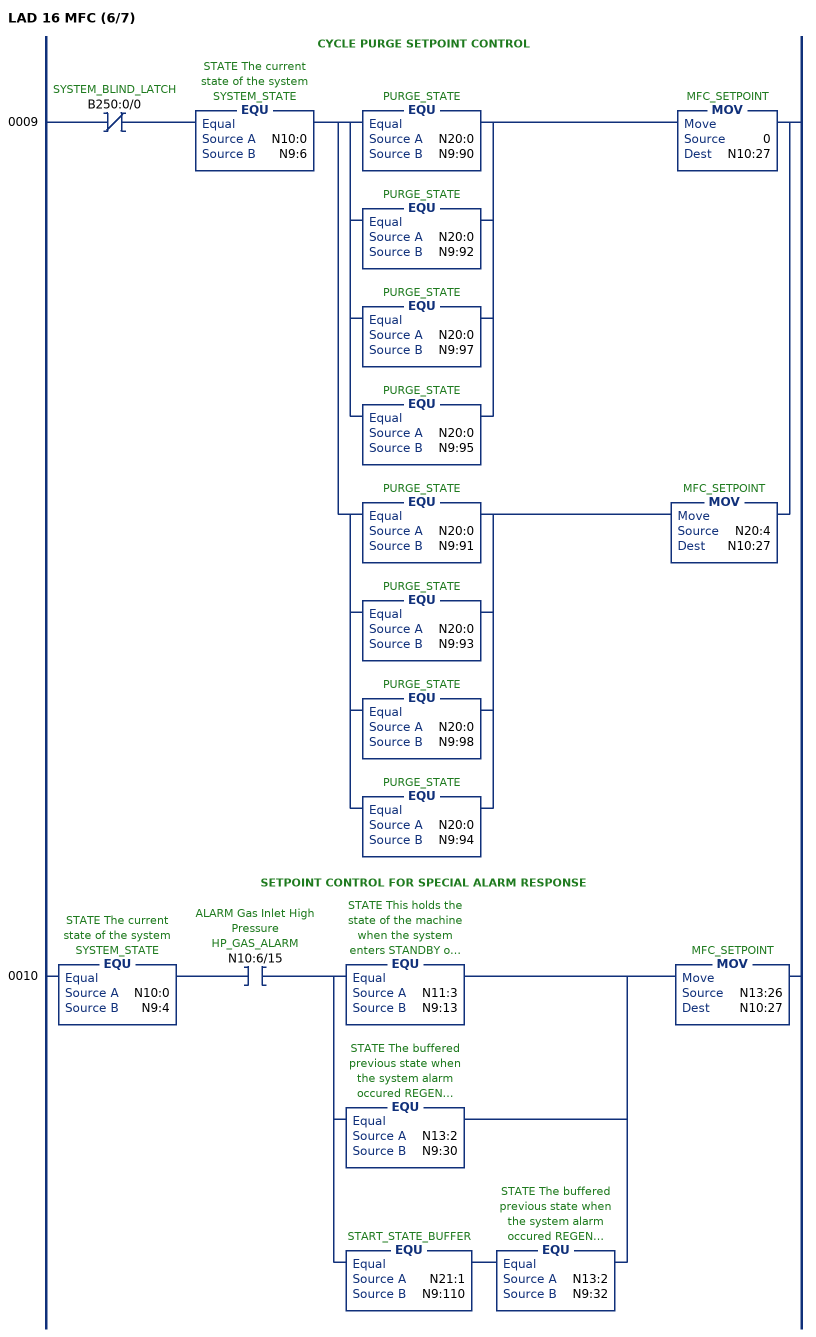
% Rung: 9 %
% TITLE: CYCLE PURGE SETPOINT CONTROL %
SOR XIO B250:0/0 EQU N10:0 N9:6 BST BST EQU N20:0 N9:90 NXB EQU N20:0 N9:92 NXB EQU N20:0 N9:97 NXB EQU N20:0 N9:95 BND MOV 0 N10:27 NXB BST EQU N20:0 N9:91 NXB EQU N20:0 N9:93 NXB EQU N20:0 N9:98 NXB EQU N20:0 N9:94 BND MOV N20:4 N10:27 BND EOR
%   B250:0/0  SYSTEM_BLIND_LATCH %
%   N10:0  SYSTEM_STATE  "STATE The current state of the system" %
%   N9:6  SYSTEM_PURGE %
%   N20:0  PURGE_STATE %
%   N9:90  PURGE_IDLE %
%   N9:92  PURGE_VENT_ADSORBER %
%   N9:97  PURGE_VENT_ADS_2 %
%   N9:95  PURGE_FINAL_VENT %
%   N10:27  MFC_SETPOINT %
%   N9:91  PURGE_INIT_VENT %
%   N9:93  PURGE_VENT_GETTER %
%   N9:98  PURGE_VENT_GET_2 %
%   N9:94  PURGE_BACKFILL %
%   N20:4  PURGE_FLOW %
% Rung: 10 %
% TITLE: SETPOINT CONTROL FOR SPECIAL ALARM RESPONSE %
SOR EQU N10:0 N9:4 XIC N10:6/15 BST EQU N11:3 N9:13 NXB EQU N13:2 N9:30 NXB EQU N21:1 N9:110 EQU N13:2 N9:32 BND MOV N13:26 N10:27 EOR
%   N10:0  SYSTEM_STATE  "STATE The current state of the system" %
%   N9:4  SYSTEM_ALARM  "STATE System Alarm" %
%   N10:6/15  HP_GAS_ALARM  "ALARM Gas Inlet High Pressure" %
%   N11:3  PROC_STATE_BUFFER  "STATE This holds the state of the machine when the system enters STANDBY or ALARM" %
%   N9:13  PROC_OVERLAP  "STATE Process Purify Overlap" %
%   N13:2  REGEN_SYSTEM_BUFFER  "STATE The buffered previous state when the system alarm occured" %
%   N9:30  REGEN_STANDBY  "STATE Regen Standby" %
%   N21:1  START_STATE_BUFFER %
%   N9:110  START_REG_VENT %
%   N9:32  REGEN_VENT  "STATE Regen Vent" %
%   N13:26  REGEN_BLEED_FLOW %
%   N10:27  MFC_SETPOINT %

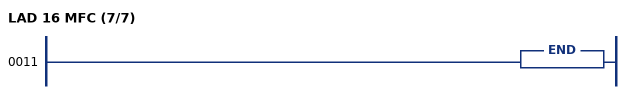
% Rung: 11 %
SOR END EOR

LADDER 17 "BYPASS"    % Controls the bypass %
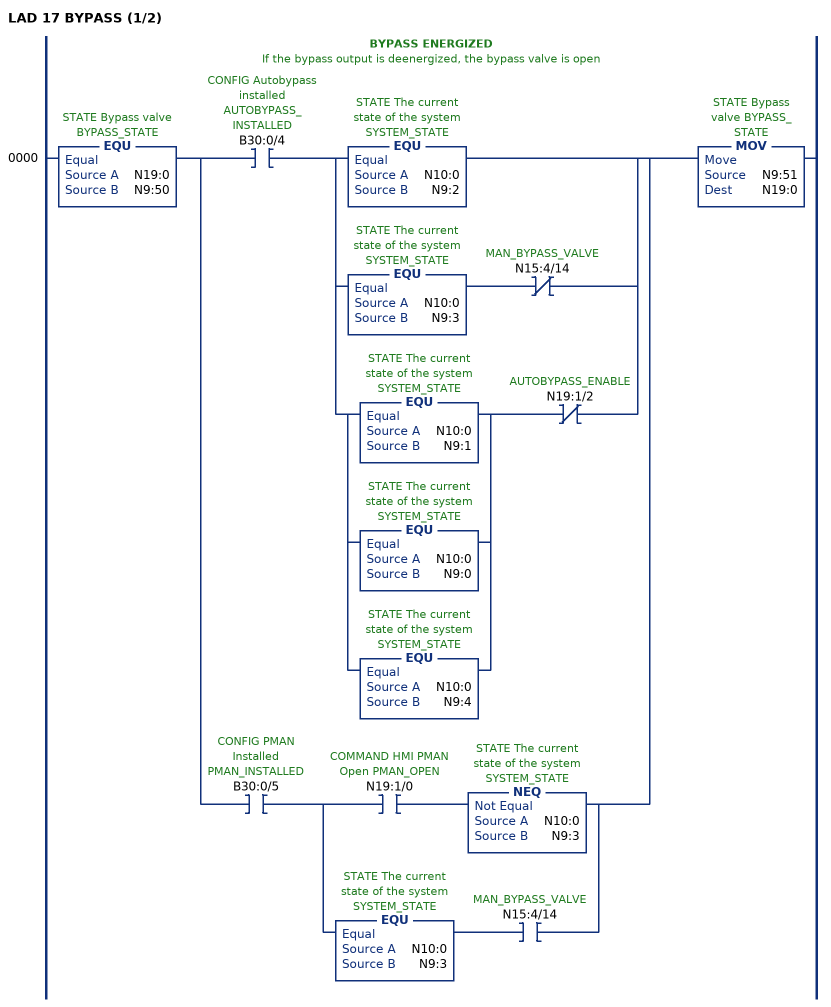
% Rung: 0 %
% TITLE: BYPASS ENERGIZED %
% If the bypass output is deenergized, the bypass valve is open %
SOR EQU N19:0 N9:50 BST XIC B30:0/4 BST EQU N10:0 N9:2 NXB EQU N10:0 N9:3 XIO N15:4/14 NXB BST EQU N10:0 N9:1 NXB EQU N10:0 N9:0 NXB EQU N10:0 N9:4 BND XIO N19:1/2 BND NXB XIC B30:0/5 BST XIC N19:1/0 NEQ N10:0 N9:3 NXB EQU N10:0 N9:3 XIC N15:4/14 BND BND MOV N9:51 N19:0 EOR
%   N19:0  BYPASS_STATE  "STATE Bypass valve" %
%   N9:50  BYPASS_DEENERGIZED  "STATE Bypass Deenergized" %
%   B30:0/4  AUTOBYPASS_INSTALLED  "CONFIG Autobypass installed" %
%   N10:0  SYSTEM_STATE  "STATE The current state of the system" %
%   N9:2  SYSTEM_PROCESS  "STATE System Process" %
%   N9:3  SYSTEM_MANUAL  "STATE System Manual" %
%   N15:4/14  MAN_BYPASS_VALVE %
%   N9:1  SYSTEM_STANDBY  "STATE System Process" %
%   N9:0  SYSTEM_OFFLINE %
%   N9:4  SYSTEM_ALARM  "STATE System Alarm" %
%   N19:1/2  AUTOBYPASS_ENABLE %
%   B30:0/5  PMAN_INSTALLED  "CONFIG PMAN Installed" %
%   N19:1/0  PMAN_OPEN  "COMMAND HMI PMAN Open" %
%   N9:51  BYPASS_ENERGIZED  "STATE Bypass Energized" %

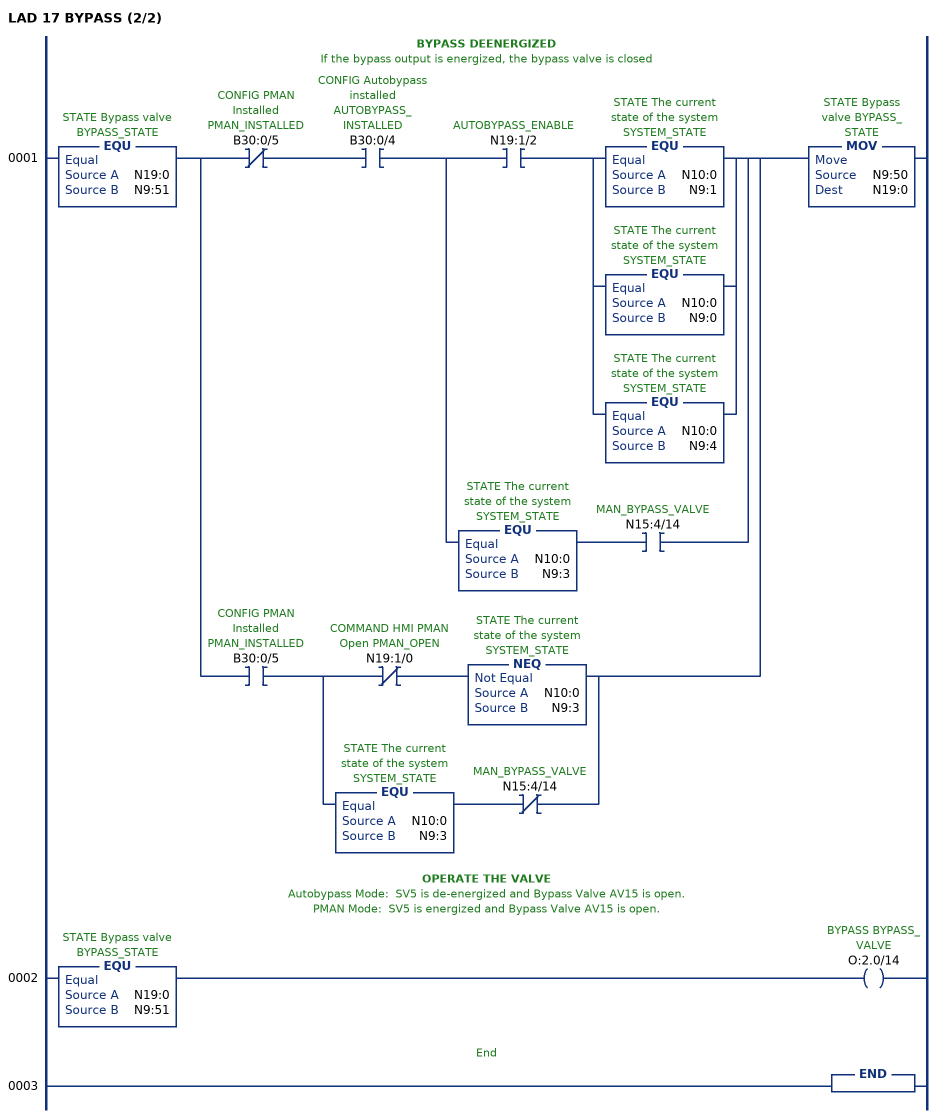
% Rung: 1 %
% TITLE: BYPASS DEENERGIZED %
% If the bypass output is energized, the bypass valve is closed %
SOR EQU N19:0 N9:51 BST XIO B30:0/5 XIC B30:0/4 BST XIC N19:1/2 BST EQU N10:0 N9:1 NXB EQU N10:0 N9:0 NXB EQU N10:0 N9:4 BND NXB EQU N10:0 N9:3 XIC N15:4/14 BND NXB XIC B30:0/5 BST XIO N19:1/0 NEQ N10:0 N9:3 NXB EQU N10:0 N9:3 XIO N15:4/14 BND BND MOV N9:50 N19:0 EOR
%   N19:0  BYPASS_STATE  "STATE Bypass valve" %
%   N9:51  BYPASS_ENERGIZED  "STATE Bypass Energized" %
%   B30:0/5  PMAN_INSTALLED  "CONFIG PMAN Installed" %
%   B30:0/4  AUTOBYPASS_INSTALLED  "CONFIG Autobypass installed" %
%   N19:1/2  AUTOBYPASS_ENABLE %
%   N10:0  SYSTEM_STATE  "STATE The current state of the system" %
%   N9:1  SYSTEM_STANDBY  "STATE System Process" %
%   N9:0  SYSTEM_OFFLINE %
%   N9:4  SYSTEM_ALARM  "STATE System Alarm" %
%   N9:3  SYSTEM_MANUAL  "STATE System Manual" %
%   N15:4/14  MAN_BYPASS_VALVE %
%   N19:1/0  PMAN_OPEN  "COMMAND HMI PMAN Open" %
%   N9:50  BYPASS_DEENERGIZED  "STATE Bypass Deenergized" %
% Rung: 2 %
% TITLE: OPERATE THE VALVE %
% Autobypass Mode:  SV5 is de-energized and Bypass Valve AV15 is open.
% PMAN Mode:  SV5 is energized and Bypass Valve AV15 is open. %
SOR EQU N19:0 N9:51 OTE O:2.0/14 EOR
%   N19:0  BYPASS_STATE  "STATE Bypass valve" %
%   N9:51  BYPASS_ENERGIZED  "STATE Bypass Energized" %
%   O:2.0/14  BYPASS_VALVE  "BYPASS" %
% Rung: 3 %
% End %
SOR END EOR

LADDER 20 "ADS A"    % Controls the Adsorber A %
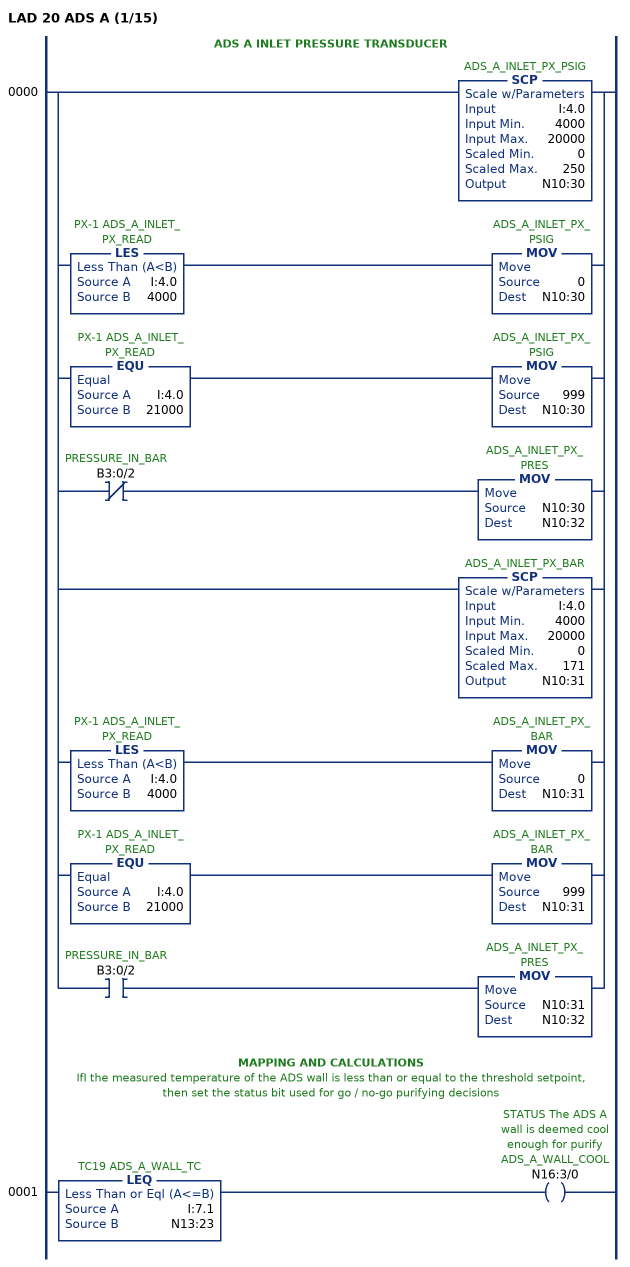
% Rung: 0 %
% TITLE: ADS A INLET PRESSURE TRANSDUCER %
SOR BST SCP I:4.0 4000 20000 0 250 N10:30 NXB LES I:4.0 4000 MOV 0 N10:30 NXB EQU I:4.0 21000 MOV 999 N10:30 NXB XIO B3:0/2 MOV N10:30 N10:32 NXB SCP I:4.0 4000 20000 0 171 N10:31 NXB LES I:4.0 4000 MOV 0 N10:31 NXB EQU I:4.0 21000 MOV 999 N10:31 NXB XIC B3:0/2 MOV N10:31 N10:32 BND EOR
%   I:4.0  ADS_A_INLET_PX_READ  "PX-1" %
%   N10:30  ADS_A_INLET_PX_PSIG %
%   B3:0/2  PRESSURE_IN_BAR %
%   N10:32  ADS_A_INLET_PX_PRES %
%   N10:31  ADS_A_INLET_PX_BAR %
% Rung: 1 %
% TITLE: MAPPING AND CALCULATIONS %
% IfI the measured temperature of the ADS wall is less than or equal to the threshold setpoint, then set the status bit used for go / no-go purifying decisions %
SOR LEQ I:7.1 N13:23 OTE N16:3/0 EOR
%   I:7.1  ADS_A_WALL_TC  "TC19" %
%   N13:23  ADS_WALL_TEMP_COOL  "CONFIG The temp at which the adsorber wall is deemed to be cool enough to purify" %
%   N16:3/0  ADS_A_WALL_COOL  "STATUS The ADS A wall is deemed cool enough for purify" %

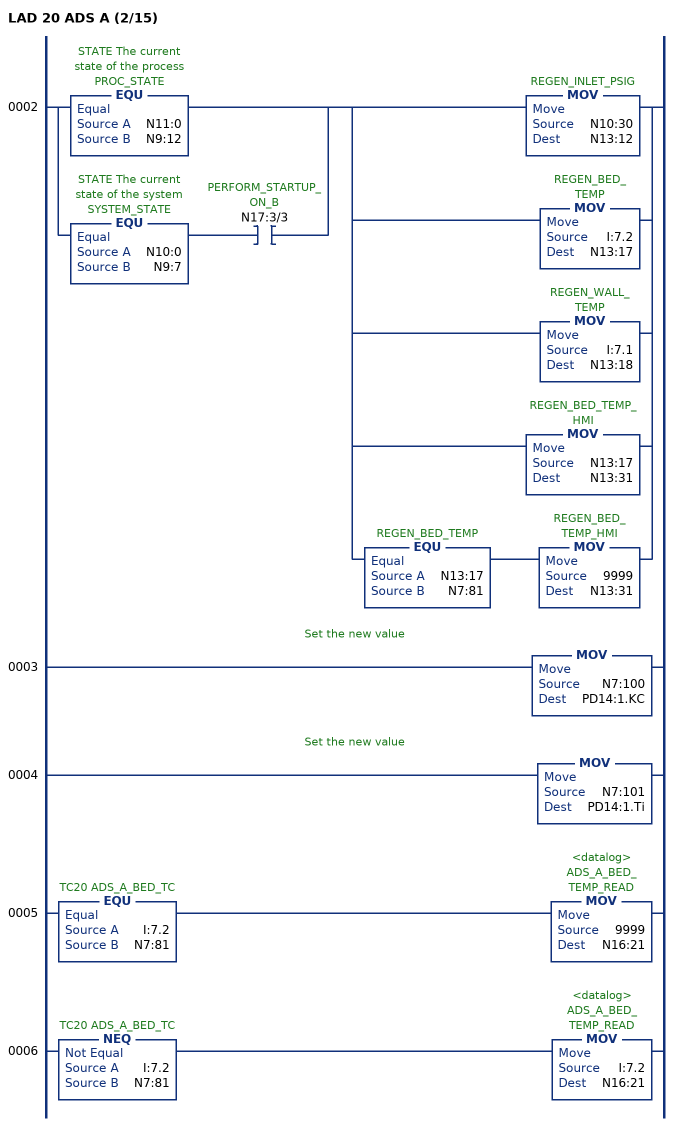
% Rung: 2 %
SOR BST EQU N11:0 N9:12 NXB EQU N10:0 N9:7 XIC N17:3/3 BND BST MOV N10:30 N13:12 NXB MOV I:7.2 N13:17 NXB MOV I:7.1 N13:18 NXB MOV N13:17 N13:31 NXB EQU N13:17 N7:81 MOV 9999 N13:31 BND EOR
%   N11:0  PROC_STATE  "STATE The current state of the process" %
%   N9:12  PROC_PFY_B_REG_A  "STATE Process Purify B" %
%   N10:0  SYSTEM_STATE  "STATE The current state of the system" %
%   N9:7  SYSTEM_COLD_START %
%   N17:3/3  PERFORM_STARTUP_ON_B %
%   N10:30  ADS_A_INLET_PX_PSIG %
%   N13:12  REGEN_INLET_PSIG %
%   I:7.2  ADS_A_BED_TC  "TC20" %
%   N13:17  REGEN_BED_TEMP %
%   I:7.1  ADS_A_WALL_TC  "TC19" %
%   N13:18  REGEN_WALL_TEMP %
%   N13:31  REGEN_BED_TEMP_HMI %
%   N7:81  TC_OPEN_SP  "CONFIG The value read by an open TC input" %
% Rung: 3 %
% Set the new value %
SOR MOV N7:100 PD14:1.KC EOR
%   N7:100  BLANKET_P  "CONFIG Blanket Proportional Gain New" %
% Rung: 4 %
% Set the new value %
SOR MOV N7:101 PD14:1.Ti EOR
%   N7:101  BLANKET_I  "CONFIG Blanket Integral Gain New" %
% Rung: 5 %
SOR EQU I:7.2 N7:81 MOV 9999 N16:21 EOR
%   I:7.2  ADS_A_BED_TC  "TC20" %
%   N7:81  TC_OPEN_SP  "CONFIG The value read by an open TC input" %
%   N16:21  ADS_A_BED_TEMP_READ  "<datalog>" %
% Rung: 6 %
SOR NEQ I:7.2 N7:81 MOV I:7.2 N16:21 EOR
%   I:7.2  ADS_A_BED_TC  "TC20" %
%   N7:81  TC_OPEN_SP  "CONFIG The value read by an open TC input" %
%   N16:21  ADS_A_BED_TEMP_READ  "<datalog>" %

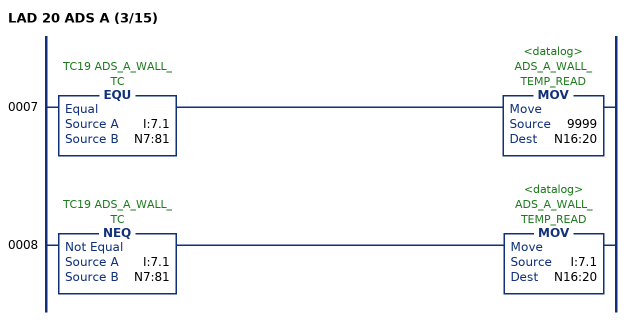
% Rung: 7 %
SOR EQU I:7.1 N7:81 MOV 9999 N16:20 EOR
%   I:7.1  ADS_A_WALL_TC  "TC19" %
%   N7:81  TC_OPEN_SP  "CONFIG The value read by an open TC input" %
%   N16:20  ADS_A_WALL_TEMP_READ  "<datalog>" %
% Rung: 8 %
SOR NEQ I:7.1 N7:81 MOV I:7.1 N16:20 EOR
%   I:7.1  ADS_A_WALL_TC  "TC19" %
%   N7:81  TC_OPEN_SP  "CONFIG The value read by an open TC input" %
%   N16:20  ADS_A_WALL_TEMP_READ  "<datalog>" %

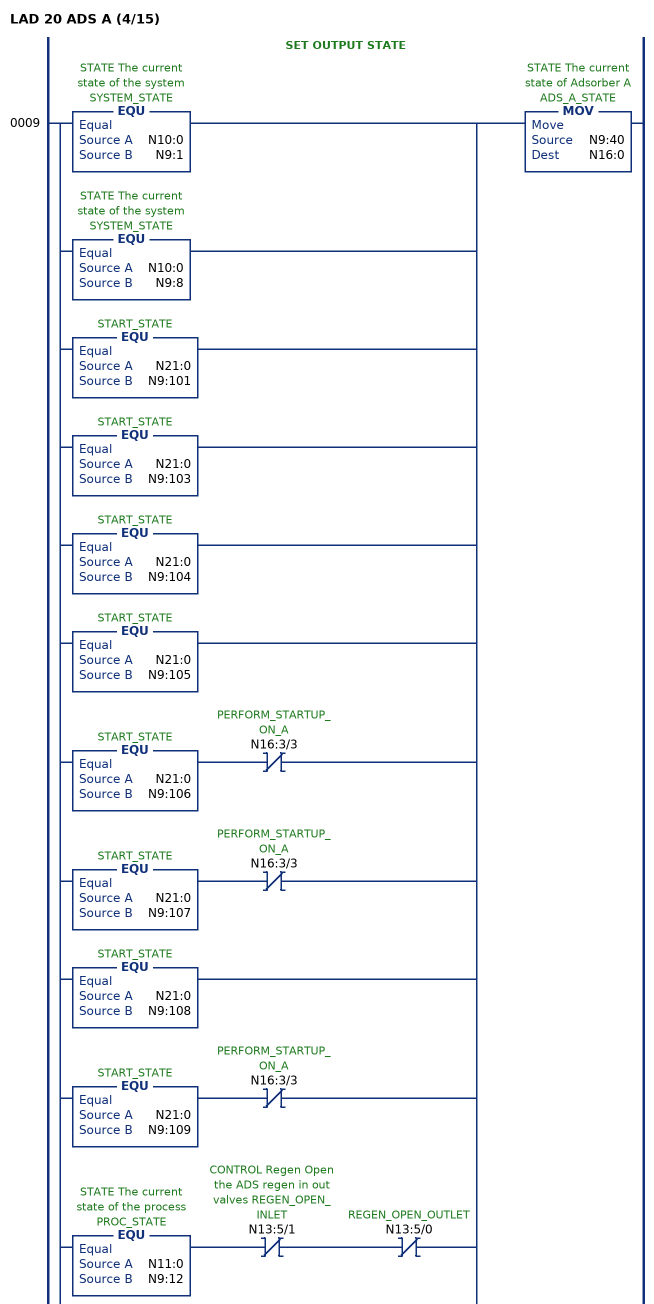

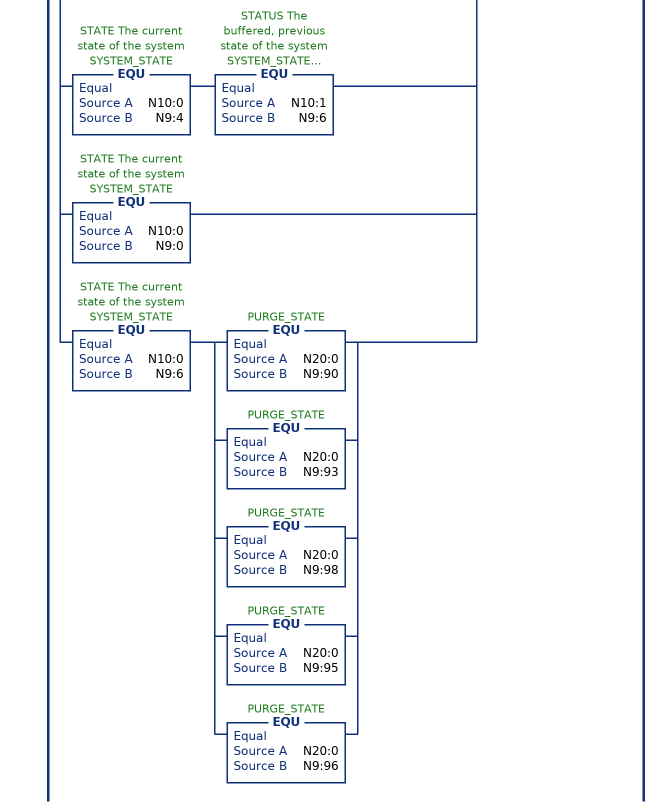
% Rung: 9 %
% TITLE: SET OUTPUT STATE %
SOR BST EQU N10:0 N9:1 NXB EQU N10:0 N9:8 NXB BST EQU N21:0 N9:101 NXB EQU N21:0 N9:103 NXB EQU N21:0 N9:104 NXB EQU N21:0 N9:105 NXB EQU N21:0 N9:106 XIO N16:3/3 NXB EQU N21:0 N9:107 XIO N16:3/3 NXB EQU N21:0 N9:108 NXB EQU N21:0 N9:109 XIO N16:3/3 BND NXB EQU N11:0 N9:12 XIO N13:5/1 XIO N13:5/0 NXB EQU N10:0 N9:4 EQU N10:1 N9:6 NXB EQU N10:0 N9:0 NXB EQU N10:0 N9:6 BST EQU N20:0 N9:90 NXB EQU N20:0 N9:93 NXB EQU N20:0 N9:98 NXB EQU N20:0 N9:95 NXB EQU N20:0 N9:96 BND BND MOV N9:40 N16:0 EOR
%   N10:0  SYSTEM_STATE  "STATE The current state of the system" %
%   N9:1  SYSTEM_STANDBY  "STATE System Process" %
%   N9:8  SYSTEM_SUPPLEMENTAL %
%   N21:0  START_STATE %
%   N9:101  START_COOL %
%   N9:103  START_VENT_GET_1 %
%   N9:104  START_HEAT %
%   N9:105  START_VENT_ALL %
%   N9:106  START_BACKFILL_1 %
%   N16:3/3  PERFORM_STARTUP_ON_A %
%   N9:107  START_VENT_ADS_2 %
%   N9:108  START_VENT_GET_2 %
%   N9:109  START_BACKFILL_2 %
%   N11:0  PROC_STATE  "STATE The current state of the process" %
%   N9:12  PROC_PFY_B_REG_A  "STATE Process Purify B" %
%   N13:5/1  REGEN_OPEN_INLET  "CONTROL Regen Open the ADS regen in out valves" %
%   N13:5/0  REGEN_OPEN_OUTLET %
%   N9:4  SYSTEM_ALARM  "STATE System Alarm" %
%   N10:1  SYSTEM_STATE_BUFFER  "STATUS The buffered, previous state of the system" %
%   N9:6  SYSTEM_PURGE %
%   N9:0  SYSTEM_OFFLINE %
%   N20:0  PURGE_STATE %
%   N9:90  PURGE_IDLE %
%   N9:93  PURGE_VENT_GETTER %
%   N9:98  PURGE_VENT_GET_2 %
%   N9:95  PURGE_FINAL_VENT %
%   N9:96  PURGE_DONE %
%   N9:40  ADS_STANDBY  "STATE ADS Standby" %
%   N16:0  ADS_A_STATE  "STATE The current state of Adsorber A" %

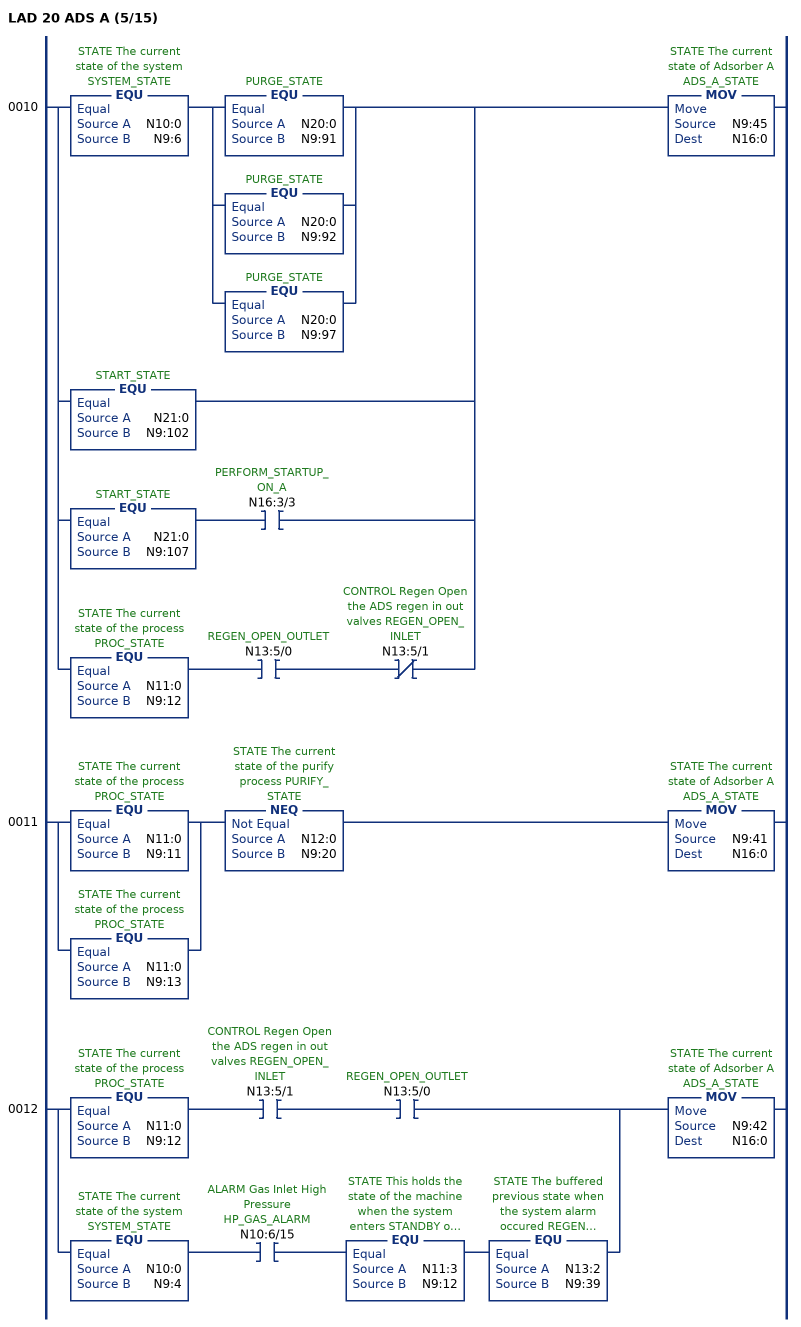
% Rung: 10 %
SOR BST EQU N10:0 N9:6 BST EQU N20:0 N9:91 NXB EQU N20:0 N9:92 NXB EQU N20:0 N9:97 BND NXB BST EQU N21:0 N9:102 NXB EQU N21:0 N9:107 XIC N16:3/3 BND NXB EQU N11:0 N9:12 XIC N13:5/0 XIO N13:5/1 BND MOV N9:45 N16:0 EOR
%   N10:0  SYSTEM_STATE  "STATE The current state of the system" %
%   N9:6  SYSTEM_PURGE %
%   N20:0  PURGE_STATE %
%   N9:91  PURGE_INIT_VENT %
%   N9:92  PURGE_VENT_ADSORBER %
%   N9:97  PURGE_VENT_ADS_2 %
%   N21:0  START_STATE %
%   N9:102  START_VENT_ADS_1 %
%   N9:107  START_VENT_ADS_2 %
%   N16:3/3  PERFORM_STARTUP_ON_A %
%   N11:0  PROC_STATE  "STATE The current state of the process" %
%   N9:12  PROC_PFY_B_REG_A  "STATE Process Purify B" %
%   N13:5/0  REGEN_OPEN_OUTLET %
%   N13:5/1  REGEN_OPEN_INLET  "CONTROL Regen Open the ADS regen in out valves" %
%   N9:45  ADS_VENT %
%   N16:0  ADS_A_STATE  "STATE The current state of Adsorber A" %
% Rung: 11 %
SOR BST EQU N11:0 N9:11 NXB EQU N11:0 N9:13 BND NEQ N12:0 N9:20 MOV N9:41 N16:0 EOR
%   N11:0  PROC_STATE  "STATE The current state of the process" %
%   N9:11  PROC_PFY_A_REG_B  "STATE Process Purify A" %
%   N9:13  PROC_OVERLAP  "STATE Process Purify Overlap" %
%   N12:0  PURIFY_STATE  "STATE The current state of the purify process" %
%   N9:20  PURIFY_STANDBY  "STATE Purify Standby" %
%   N9:41  ADS_PURIFY  "STATE ADS Purify" %
%   N16:0  ADS_A_STATE  "STATE The current state of Adsorber A" %
% Rung: 12 %
SOR BST EQU N11:0 N9:12 XIC N13:5/1 XIC N13:5/0 NXB EQU N10:0 N9:4 XIC N10:6/15 EQU N11:3 N9:12 EQU N13:2 N9:39 BND MOV N9:42 N16:0 EOR
%   N11:0  PROC_STATE  "STATE The current state of the process" %
%   N9:12  PROC_PFY_B_REG_A  "STATE Process Purify B" %
%   N13:5/1  REGEN_OPEN_INLET  "CONTROL Regen Open the ADS regen in out valves" %
%   N13:5/0  REGEN_OPEN_OUTLET %
%   N10:0  SYSTEM_STATE  "STATE The current state of the system" %
%   N9:4  SYSTEM_ALARM  "STATE System Alarm" %
%   N10:6/15  HP_GAS_ALARM  "ALARM Gas Inlet High Pressure" %
%   N11:3  PROC_STATE_BUFFER  "STATE This holds the state of the machine when the system enters STANDBY or ALARM" %
%   N13:2  REGEN_SYSTEM_BUFFER  "STATE The buffered previous state when the system alarm occured" %
%   N9:39  REGEN_BACKFILL %
%   N9:42  ADS_REGEN  "STATE ADS Regen" %
%   N16:0  ADS_A_STATE  "STATE The current state of Adsorber A" %

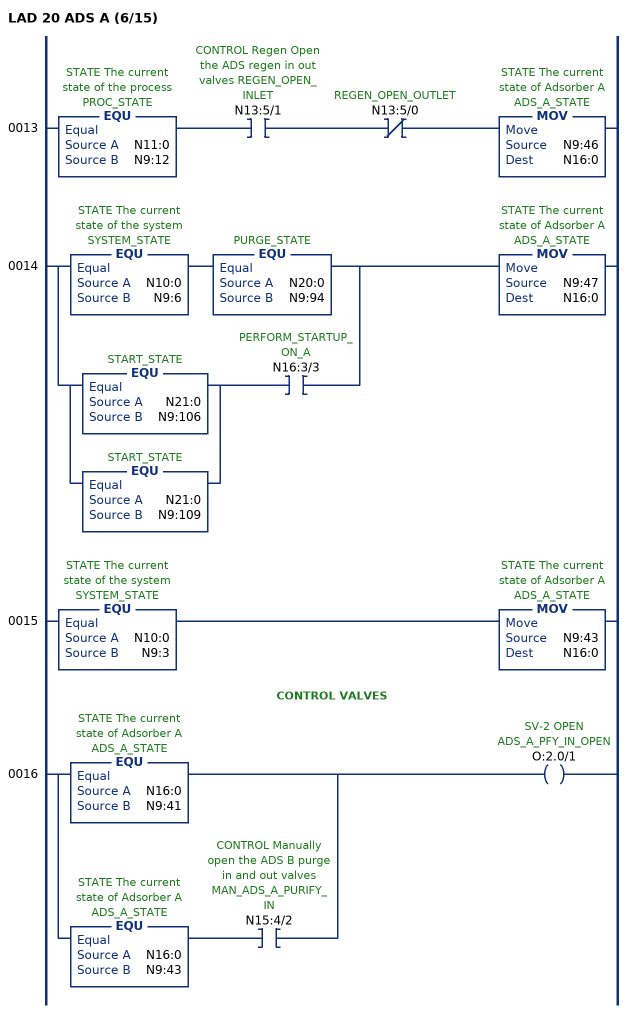
% Rung: 13 %
SOR EQU N11:0 N9:12 XIC N13:5/1 XIO N13:5/0 MOV N9:46 N16:0 EOR
%   N11:0  PROC_STATE  "STATE The current state of the process" %
%   N9:12  PROC_PFY_B_REG_A  "STATE Process Purify B" %
%   N13:5/1  REGEN_OPEN_INLET  "CONTROL Regen Open the ADS regen in out valves" %
%   N13:5/0  REGEN_OPEN_OUTLET %
%   N9:46  ADS_REGEN_BACKFILL %
%   N16:0  ADS_A_STATE  "STATE The current state of Adsorber A" %
% Rung: 14 %
SOR BST EQU N10:0 N9:6 EQU N20:0 N9:94 NXB BST EQU N21:0 N9:106 NXB EQU N21:0 N9:109 BND XIC N16:3/3 BND MOV N9:47 N16:0 EOR
%   N10:0  SYSTEM_STATE  "STATE The current state of the system" %
%   N9:6  SYSTEM_PURGE %
%   N20:0  PURGE_STATE %
%   N9:94  PURGE_BACKFILL %
%   N21:0  START_STATE %
%   N9:106  START_BACKFILL_1 %
%   N9:109  START_BACKFILL_2 %
%   N16:3/3  PERFORM_STARTUP_ON_A %
%   N9:47  ADS_BACKFILL %
%   N16:0  ADS_A_STATE  "STATE The current state of Adsorber A" %
% Rung: 15 %
SOR EQU N10:0 N9:3 MOV N9:43 N16:0 EOR
%   N10:0  SYSTEM_STATE  "STATE The current state of the system" %
%   N9:3  SYSTEM_MANUAL  "STATE System Manual" %
%   N9:43  ADS_MANUAL  "STATE ADS Manual" %
%   N16:0  ADS_A_STATE  "STATE The current state of Adsorber A" %
% Rung: 16 %
% TITLE: CONTROL VALVES %
SOR BST EQU N16:0 N9:41 NXB EQU N16:0 N9:43 XIC N15:4/2 BND OTE O:2.0/1 EOR
%   N16:0  ADS_A_STATE  "STATE The current state of Adsorber A" %
%   N9:41  ADS_PURIFY  "STATE ADS Purify" %
%   N9:43  ADS_MANUAL  "STATE ADS Manual" %
%   N15:4/2  MAN_ADS_A_PURIFY_IN  "CONTROL Manually open the ADS B purge in and out valves" %
%   O:2.0/1  ADS_A_PFY_IN_OPEN  "SV-2 OPEN" %

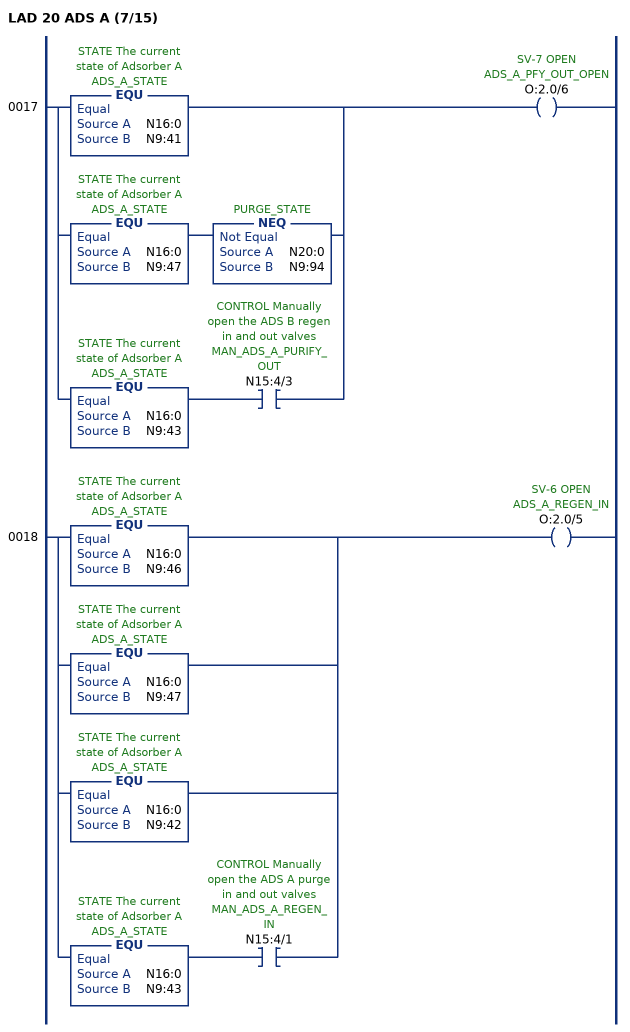
% Rung: 17 %
SOR BST EQU N16:0 N9:41 NXB EQU N16:0 N9:47 NEQ N20:0 N9:94 NXB EQU N16:0 N9:43 XIC N15:4/3 BND OTE O:2.0/6 EOR
%   N16:0  ADS_A_STATE  "STATE The current state of Adsorber A" %
%   N9:41  ADS_PURIFY  "STATE ADS Purify" %
%   N9:47  ADS_BACKFILL %
%   N20:0  PURGE_STATE %
%   N9:94  PURGE_BACKFILL %
%   N9:43  ADS_MANUAL  "STATE ADS Manual" %
%   N15:4/3  MAN_ADS_A_PURIFY_OUT  "CONTROL Manually open the ADS B regen in and out valves" %
%   O:2.0/6  ADS_A_PFY_OUT_OPEN  "SV-7 OPEN" %
% Rung: 18 %
SOR BST EQU N16:0 N9:46 NXB EQU N16:0 N9:47 NXB EQU N16:0 N9:42 NXB EQU N16:0 N9:43 XIC N15:4/1 BND OTE O:2.0/5 EOR
%   N16:0  ADS_A_STATE  "STATE The current state of Adsorber A" %
%   N9:46  ADS_REGEN_BACKFILL %
%   N9:47  ADS_BACKFILL %
%   N9:42  ADS_REGEN  "STATE ADS Regen" %
%   N9:43  ADS_MANUAL  "STATE ADS Manual" %
%   N15:4/1  MAN_ADS_A_REGEN_IN  "CONTROL Manually open the ADS A purge in and out valves" %
%   O:2.0/5  ADS_A_REGEN_IN  "SV-6 OPEN" %

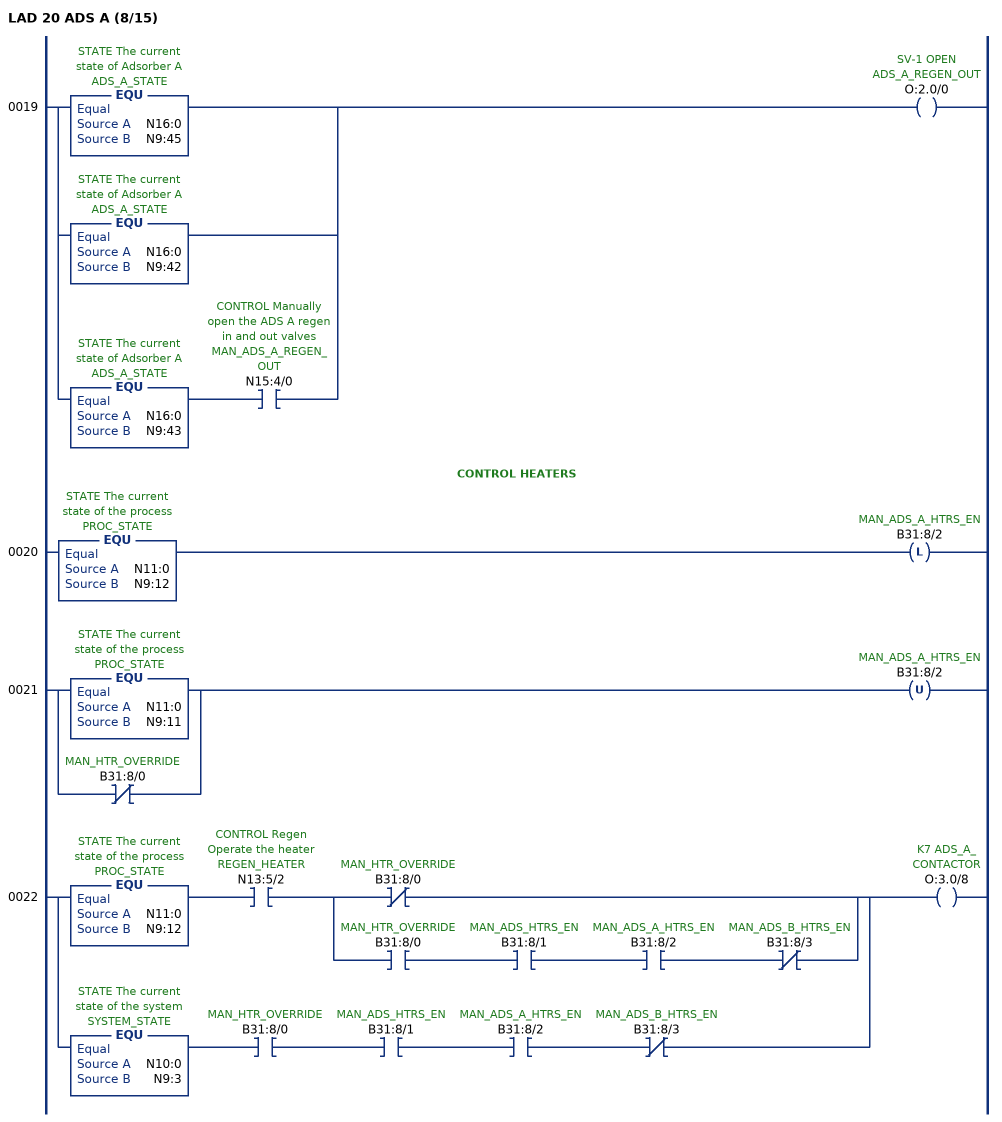
% Rung: 19 %
SOR BST EQU N16:0 N9:45 NXB EQU N16:0 N9:42 NXB EQU N16:0 N9:43 XIC N15:4/0 BND OTE O:2.0/0 EOR
%   N16:0  ADS_A_STATE  "STATE The current state of Adsorber A" %
%   N9:45  ADS_VENT %
%   N9:42  ADS_REGEN  "STATE ADS Regen" %
%   N9:43  ADS_MANUAL  "STATE ADS Manual" %
%   N15:4/0  MAN_ADS_A_REGEN_OUT  "CONTROL Manually open the ADS A regen in and out valves" %
%   O:2.0/0  ADS_A_REGEN_OUT  "SV-1 OPEN" %
% Rung: 20 %
% TITLE: CONTROL HEATERS %
SOR EQU N11:0 N9:12 OTL B31:8/2 EOR
%   N11:0  PROC_STATE  "STATE The current state of the process" %
%   N9:12  PROC_PFY_B_REG_A  "STATE Process Purify B" %
%   B31:8/2  MAN_ADS_A_HTRS_EN %
% Rung: 21 %
SOR BST EQU N11:0 N9:11 NXB XIO B31:8/0 BND OTU B31:8/2 EOR
%   N11:0  PROC_STATE  "STATE The current state of the process" %
%   N9:11  PROC_PFY_A_REG_B  "STATE Process Purify A" %
%   B31:8/0  MAN_HTR_OVERRIDE %
%   B31:8/2  MAN_ADS_A_HTRS_EN %
% Rung: 22 %
SOR BST EQU N11:0 N9:12 XIC N13:5/2 BST XIO B31:8/0 NXB XIC B31:8/0 XIC B31:8/1 XIC B31:8/2 XIO B31:8/3 BND NXB EQU N10:0 N9:3 XIC B31:8/0 XIC B31:8/1 XIC B31:8/2 XIO B31:8/3 BND OTE O:3.0/8 EOR
%   N11:0  PROC_STATE  "STATE The current state of the process" %
%   N9:12  PROC_PFY_B_REG_A  "STATE Process Purify B" %
%   N13:5/2  REGEN_HEATER  "CONTROL Regen Operate the heater" %
%   B31:8/0  MAN_HTR_OVERRIDE %
%   B31:8/1  MAN_ADS_HTRS_EN %
%   B31:8/2  MAN_ADS_A_HTRS_EN %
%   B31:8/3  MAN_ADS_B_HTRS_EN %
%   N10:0  SYSTEM_STATE  "STATE The current state of the system" %
%   N9:3  SYSTEM_MANUAL  "STATE System Manual" %
%   O:3.0/8  ADS_A_CONTACTOR  "K7" %

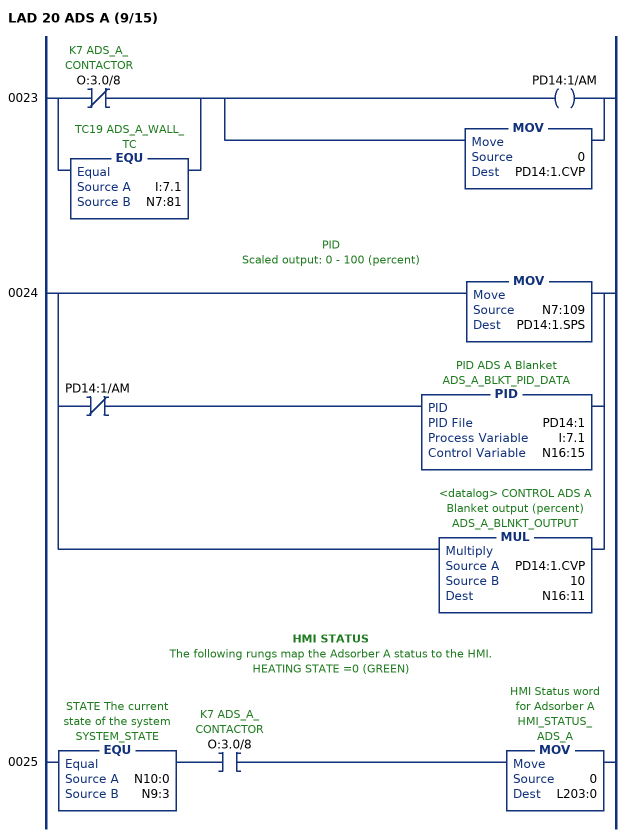
% Rung: 23 %
SOR BST XIO O:3.0/8 NXB EQU I:7.1 N7:81 BND BST OTE PD14:1/AM NXB MOV 0 PD14:1.CVP BND EOR
%   O:3.0/8  ADS_A_CONTACTOR  "K7" %
%   I:7.1  ADS_A_WALL_TC  "TC19" %
%   N7:81  TC_OPEN_SP  "CONFIG The value read by an open TC input" %
% Rung: 24 %
% PID
% Scaled output: 0 - 100 (percent) %
SOR BST MOV N7:109 PD14:1.SPS NXB XIO PD14:1/AM PID PD14:1 I:7.1 N16:15 NXB MUL PD14:1.CVP 10 N16:11 BND EOR
%   N7:109  BLANKET_SP  "<datalog> CONTROL Blanket PID Setpoint" %
%   PD14:1  ADS_A_BLKT_PID_DATA  "PID ADS A Blanket" %
%   I:7.1  ADS_A_WALL_TC  "TC19" %
%   N16:15  ADS_A_BLKT_OUTPT_RAW  "CONTROL ADS A Blanket PID Output Raw" %
%   N16:11  ADS_A_BLNKT_OUTPUT  "<datalog> CONTROL ADS A Blanket output (percent)" %
% Rung: 25 %
% TITLE: HMI STATUS %
% The following rungs map the Adsorber A status to the HMI.
% HEATING STATE =0 (GREEN) %
SOR EQU N10:0 N9:3 XIC O:3.0/8 MOV 0 L203:0 EOR
%   N10:0  SYSTEM_STATE  "STATE The current state of the system" %
%   N9:3  SYSTEM_MANUAL  "STATE System Manual" %
%   O:3.0/8  ADS_A_CONTACTOR  "K7" %
%   L203:0  HMI_STATUS_ADS_A  "HMI Status word for Adsorber A" %

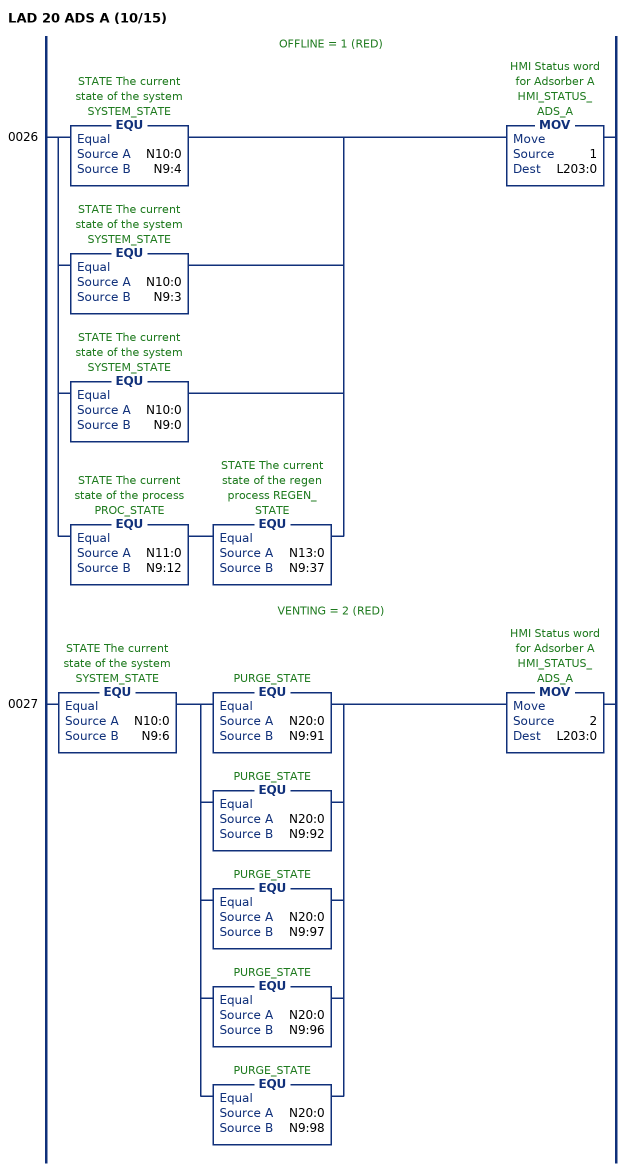
% Rung: 26 %
% OFFLINE = 1 (RED) %
SOR BST BST EQU N10:0 N9:4 NXB EQU N10:0 N9:3 NXB EQU N10:0 N9:0 BND NXB EQU N11:0 N9:12 EQU N13:0 N9:37 BND MOV 1 L203:0 EOR
%   N10:0  SYSTEM_STATE  "STATE The current state of the system" %
%   N9:4  SYSTEM_ALARM  "STATE System Alarm" %
%   N9:3  SYSTEM_MANUAL  "STATE System Manual" %
%   N9:0  SYSTEM_OFFLINE %
%   N11:0  PROC_STATE  "STATE The current state of the process" %
%   N9:12  PROC_PFY_B_REG_A  "STATE Process Purify B" %
%   N13:0  REGEN_STATE  "STATE The current state of the regen process" %
%   N9:37  REGEN_ALARM  "STATE Regen Alarm" %
%   L203:0  HMI_STATUS_ADS_A  "HMI Status word for Adsorber A" %
% Rung: 27 %
% VENTING = 2 (RED) %
SOR EQU N10:0 N9:6 BST EQU N20:0 N9:91 NXB EQU N20:0 N9:92 NXB EQU N20:0 N9:97 NXB EQU N20:0 N9:96 NXB EQU N20:0 N9:98 BND MOV 2 L203:0 EOR
%   N10:0  SYSTEM_STATE  "STATE The current state of the system" %
%   N9:6  SYSTEM_PURGE %
%   N20:0  PURGE_STATE %
%   N9:91  PURGE_INIT_VENT %
%   N9:92  PURGE_VENT_ADSORBER %
%   N9:97  PURGE_VENT_ADS_2 %
%   N9:96  PURGE_DONE %
%   N9:98  PURGE_VENT_GET_2 %
%   L203:0  HMI_STATUS_ADS_A  "HMI Status word for Adsorber A" %

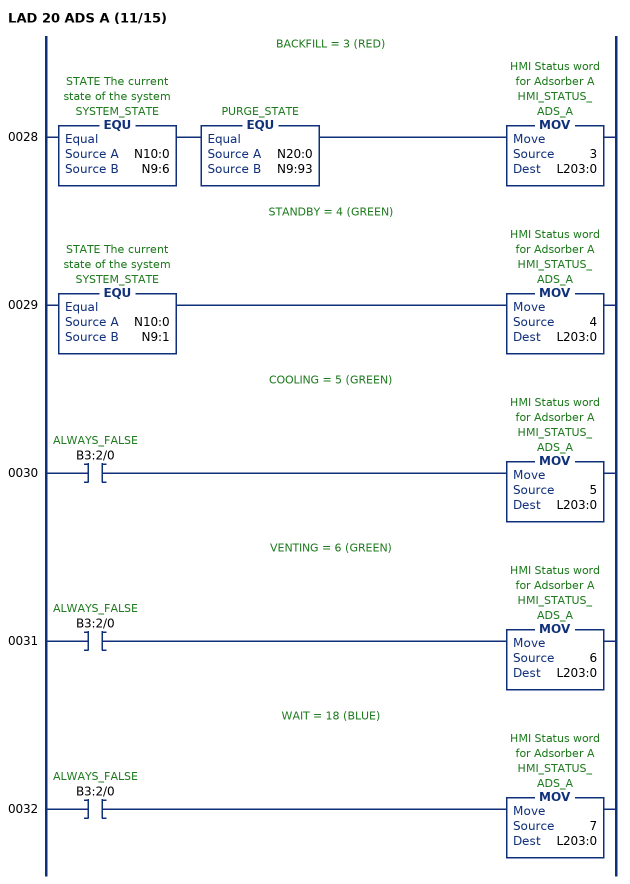
% Rung: 28 %
% BACKFILL = 3 (RED) %
SOR EQU N10:0 N9:6 EQU N20:0 N9:93 MOV 3 L203:0 EOR
%   N10:0  SYSTEM_STATE  "STATE The current state of the system" %
%   N9:6  SYSTEM_PURGE %
%   N20:0  PURGE_STATE %
%   N9:93  PURGE_VENT_GETTER %
%   L203:0  HMI_STATUS_ADS_A  "HMI Status word for Adsorber A" %
% Rung: 29 %
% STANDBY = 4 (GREEN) %
SOR EQU N10:0 N9:1 MOV 4 L203:0 EOR
%   N10:0  SYSTEM_STATE  "STATE The current state of the system" %
%   N9:1  SYSTEM_STANDBY  "STATE System Process" %
%   L203:0  HMI_STATUS_ADS_A  "HMI Status word for Adsorber A" %
% Rung: 30 %
% COOLING = 5 (GREEN) %
SOR XIC B3:2/0 MOV 5 L203:0 EOR
%   B3:2/0  ALWAYS_FALSE %
%   L203:0  HMI_STATUS_ADS_A  "HMI Status word for Adsorber A" %
% Rung: 31 %
% VENTING = 6 (GREEN) %
SOR XIC B3:2/0 MOV 6 L203:0 EOR
%   B3:2/0  ALWAYS_FALSE %
%   L203:0  HMI_STATUS_ADS_A  "HMI Status word for Adsorber A" %
% Rung: 32 %
% WAIT = 18 (BLUE) %
SOR XIC B3:2/0 MOV 7 L203:0 EOR
%   B3:2/0  ALWAYS_FALSE %
%   L203:0  HMI_STATUS_ADS_A  "HMI Status word for Adsorber A" %

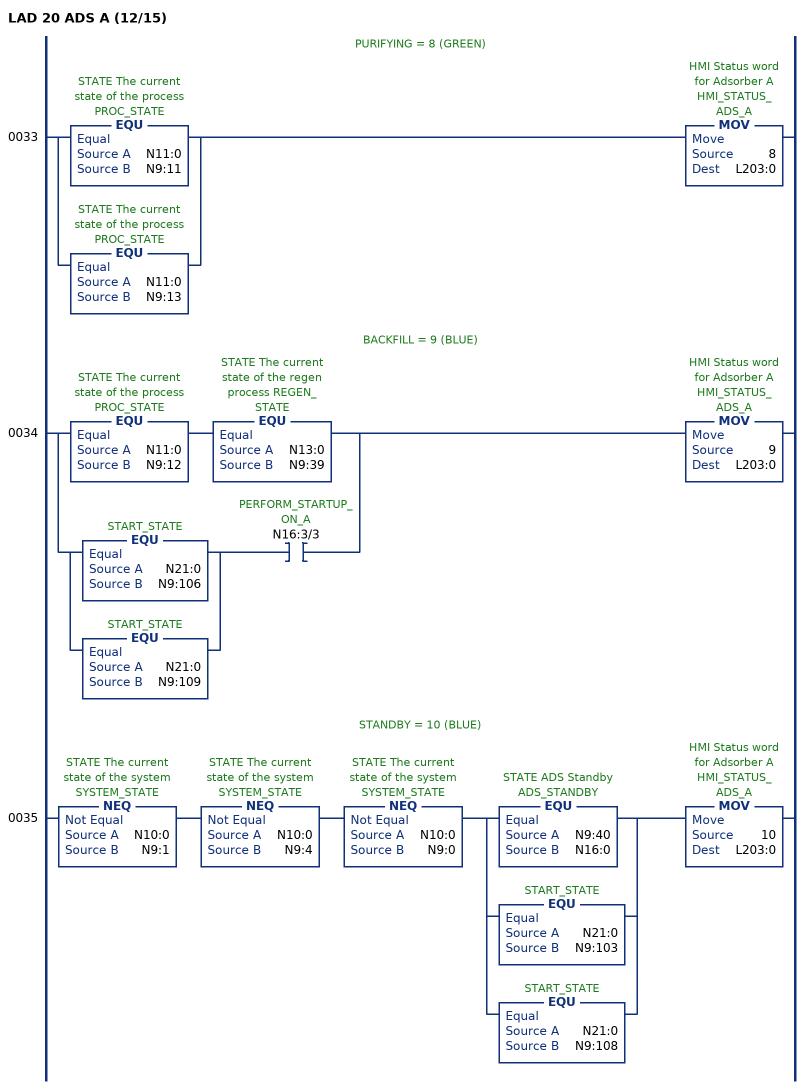
% Rung: 33 %
% PURIFYING = 8 (GREEN) %
SOR BST EQU N11:0 N9:11 NXB EQU N11:0 N9:13 BND MOV 8 L203:0 EOR
%   N11:0  PROC_STATE  "STATE The current state of the process" %
%   N9:11  PROC_PFY_A_REG_B  "STATE Process Purify A" %
%   N9:13  PROC_OVERLAP  "STATE Process Purify Overlap" %
%   L203:0  HMI_STATUS_ADS_A  "HMI Status word for Adsorber A" %
% Rung: 34 %
% BACKFILL = 9 (BLUE) %
SOR BST EQU N11:0 N9:12 EQU N13:0 N9:39 NXB BST EQU N21:0 N9:106 NXB EQU N21:0 N9:109 BND XIC N16:3/3 BND MOV 9 L203:0 EOR
%   N11:0  PROC_STATE  "STATE The current state of the process" %
%   N9:12  PROC_PFY_B_REG_A  "STATE Process Purify B" %
%   N13:0  REGEN_STATE  "STATE The current state of the regen process" %
%   N9:39  REGEN_BACKFILL %
%   N21:0  START_STATE %
%   N9:106  START_BACKFILL_1 %
%   N9:109  START_BACKFILL_2 %
%   N16:3/3  PERFORM_STARTUP_ON_A %
%   L203:0  HMI_STATUS_ADS_A  "HMI Status word for Adsorber A" %
% Rung: 35 %
% STANDBY = 10 (BLUE) %
SOR NEQ N10:0 N9:1 NEQ N10:0 N9:4 NEQ N10:0 N9:0 BST EQU N9:40 N16:0 NXB EQU N21:0 N9:103 NXB EQU N21:0 N9:108 BND MOV 10 L203:0 EOR
%   N10:0  SYSTEM_STATE  "STATE The current state of the system" %
%   N9:1  SYSTEM_STANDBY  "STATE System Process" %
%   N9:4  SYSTEM_ALARM  "STATE System Alarm" %
%   N9:0  SYSTEM_OFFLINE %
%   N9:40  ADS_STANDBY  "STATE ADS Standby" %
%   N16:0  ADS_A_STATE  "STATE The current state of Adsorber A" %
%   N21:0  START_STATE %
%   N9:103  START_VENT_GET_1 %
%   N9:108  START_VENT_GET_2 %
%   L203:0  HMI_STATUS_ADS_A  "HMI Status word for Adsorber A" %

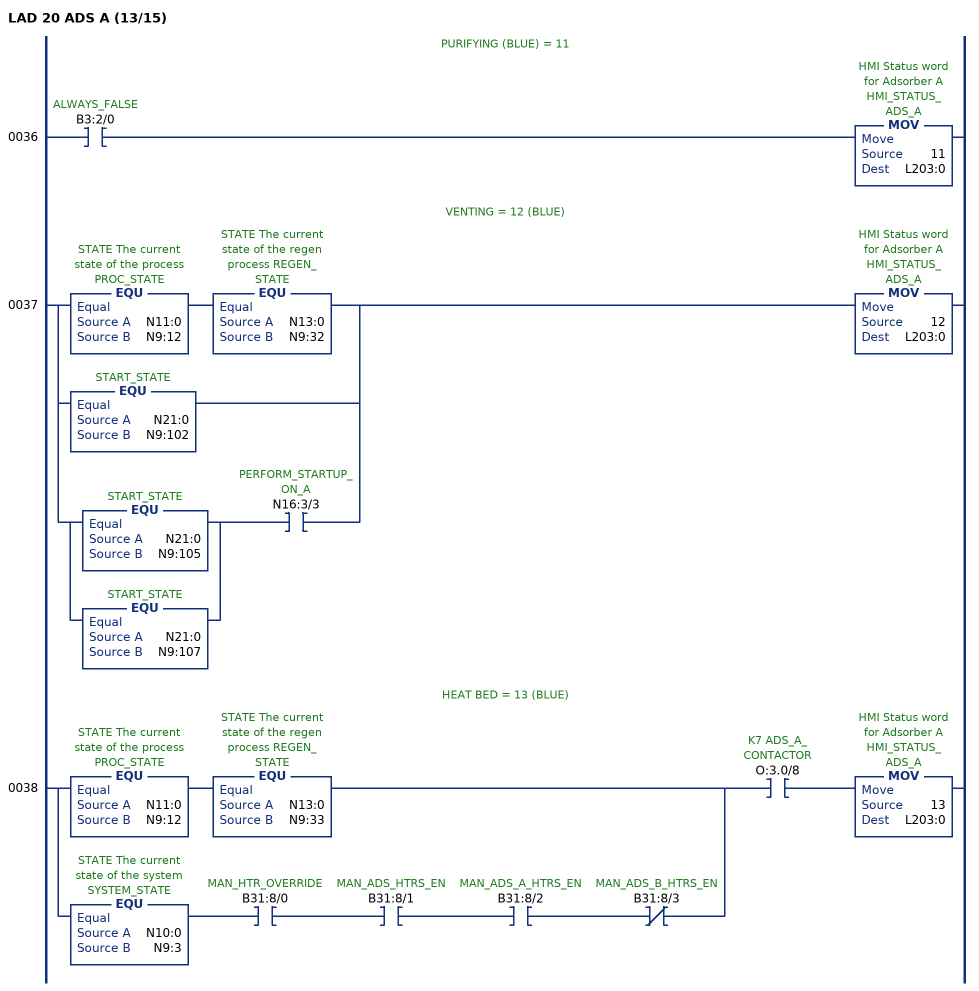
% Rung: 36 %
% PURIFYING (BLUE) = 11 %
SOR XIC B3:2/0 MOV 11 L203:0 EOR
%   B3:2/0  ALWAYS_FALSE %
%   L203:0  HMI_STATUS_ADS_A  "HMI Status word for Adsorber A" %
% Rung: 37 %
% VENTING = 12 (BLUE) %
SOR BST EQU N11:0 N9:12 EQU N13:0 N9:32 NXB BST EQU N21:0 N9:102 NXB BST EQU N21:0 N9:105 NXB EQU N21:0 N9:107 BND XIC N16:3/3 BND BND MOV 12 L203:0 EOR
%   N11:0  PROC_STATE  "STATE The current state of the process" %
%   N9:12  PROC_PFY_B_REG_A  "STATE Process Purify B" %
%   N13:0  REGEN_STATE  "STATE The current state of the regen process" %
%   N9:32  REGEN_VENT  "STATE Regen Vent" %
%   N21:0  START_STATE %
%   N9:102  START_VENT_ADS_1 %
%   N9:105  START_VENT_ALL %
%   N9:107  START_VENT_ADS_2 %
%   N16:3/3  PERFORM_STARTUP_ON_A %
%   L203:0  HMI_STATUS_ADS_A  "HMI Status word for Adsorber A" %
% Rung: 38 %
% HEAT BED = 13 (BLUE) %
SOR BST EQU N11:0 N9:12 EQU N13:0 N9:33 NXB EQU N10:0 N9:3 XIC B31:8/0 XIC B31:8/1 XIC B31:8/2 XIO B31:8/3 BND XIC O:3.0/8 MOV 13 L203:0 EOR
%   N11:0  PROC_STATE  "STATE The current state of the process" %
%   N9:12  PROC_PFY_B_REG_A  "STATE Process Purify B" %
%   N13:0  REGEN_STATE  "STATE The current state of the regen process" %
%   N9:33  REGEN_HEAT_BED  "STATE Regen Heat wall" %
%   N10:0  SYSTEM_STATE  "STATE The current state of the system" %
%   N9:3  SYSTEM_MANUAL  "STATE System Manual" %
%   B31:8/0  MAN_HTR_OVERRIDE %
%   B31:8/1  MAN_ADS_HTRS_EN %
%   B31:8/2  MAN_ADS_A_HTRS_EN %
%   B31:8/3  MAN_ADS_B_HTRS_EN %
%   O:3.0/8  ADS_A_CONTACTOR  "K7" %
%   L203:0  HMI_STATUS_ADS_A  "HMI Status word for Adsorber A" %

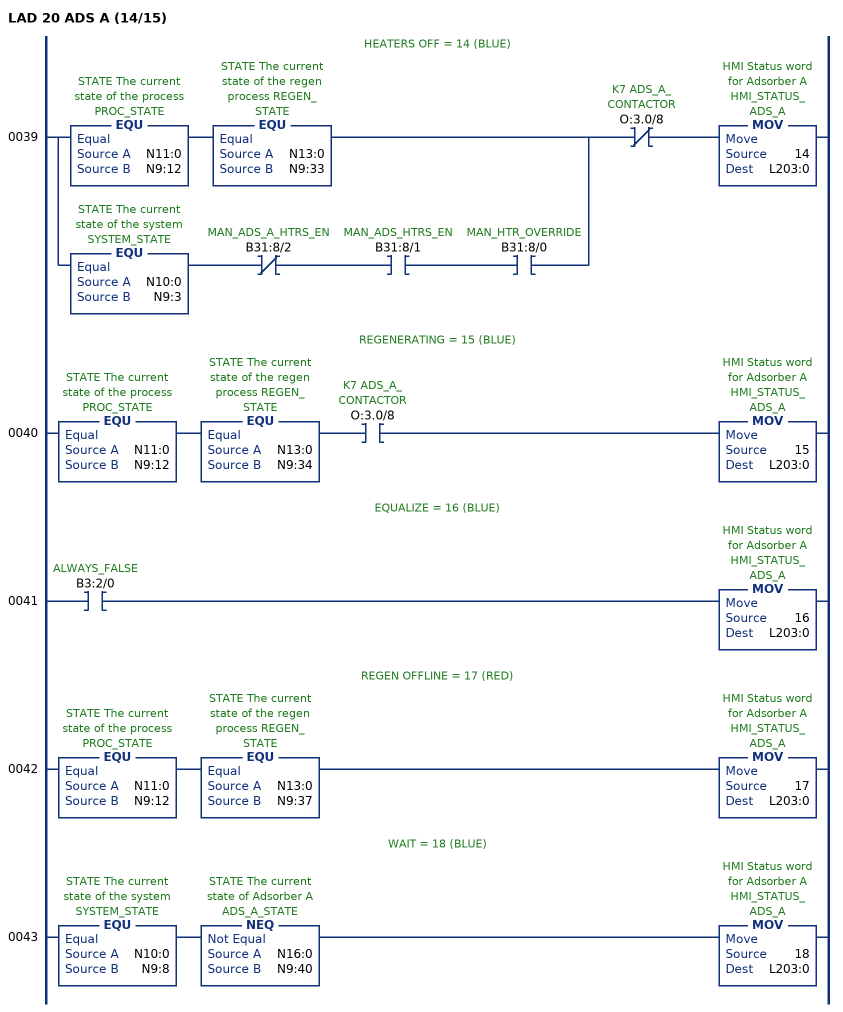
% Rung: 39 %
% HEATERS OFF = 14 (BLUE) %
SOR BST EQU N11:0 N9:12 EQU N13:0 N9:33 NXB EQU N10:0 N9:3 XIO B31:8/2 XIC B31:8/1 XIC B31:8/0 BND XIO O:3.0/8 MOV 14 L203:0 EOR
%   N11:0  PROC_STATE  "STATE The current state of the process" %
%   N9:12  PROC_PFY_B_REG_A  "STATE Process Purify B" %
%   N13:0  REGEN_STATE  "STATE The current state of the regen process" %
%   N9:33  REGEN_HEAT_BED  "STATE Regen Heat wall" %
%   N10:0  SYSTEM_STATE  "STATE The current state of the system" %
%   N9:3  SYSTEM_MANUAL  "STATE System Manual" %
%   B31:8/2  MAN_ADS_A_HTRS_EN %
%   B31:8/1  MAN_ADS_HTRS_EN %
%   B31:8/0  MAN_HTR_OVERRIDE %
%   O:3.0/8  ADS_A_CONTACTOR  "K7" %
%   L203:0  HMI_STATUS_ADS_A  "HMI Status word for Adsorber A" %
% Rung: 40 %
% REGENERATING = 15 (BLUE) %
SOR EQU N11:0 N9:12 EQU N13:0 N9:34 XIC O:3.0/8 MOV 15 L203:0 EOR
%   N11:0  PROC_STATE  "STATE The current state of the process" %
%   N9:12  PROC_PFY_B_REG_A  "STATE Process Purify B" %
%   N13:0  REGEN_STATE  "STATE The current state of the regen process" %
%   N9:34  REGEN_RUN  "STATE Regen Running" %
%   O:3.0/8  ADS_A_CONTACTOR  "K7" %
%   L203:0  HMI_STATUS_ADS_A  "HMI Status word for Adsorber A" %
% Rung: 41 %
% EQUALIZE = 16 (BLUE) %
SOR XIC B3:2/0 MOV 16 L203:0 EOR
%   B3:2/0  ALWAYS_FALSE %
%   L203:0  HMI_STATUS_ADS_A  "HMI Status word for Adsorber A" %
% Rung: 42 %
% REGEN OFFLINE = 17 (RED) %
SOR EQU N11:0 N9:12 EQU N13:0 N9:37 MOV 17 L203:0 EOR
%   N11:0  PROC_STATE  "STATE The current state of the process" %
%   N9:12  PROC_PFY_B_REG_A  "STATE Process Purify B" %
%   N13:0  REGEN_STATE  "STATE The current state of the regen process" %
%   N9:37  REGEN_ALARM  "STATE Regen Alarm" %
%   L203:0  HMI_STATUS_ADS_A  "HMI Status word for Adsorber A" %
% Rung: 43 %
% WAIT = 18 (BLUE) %
SOR EQU N10:0 N9:8 NEQ N16:0 N9:40 MOV 18 L203:0 EOR
%   N10:0  SYSTEM_STATE  "STATE The current state of the system" %
%   N9:8  SYSTEM_SUPPLEMENTAL %
%   N16:0  ADS_A_STATE  "STATE The current state of Adsorber A" %
%   N9:40  ADS_STANDBY  "STATE ADS Standby" %
%   L203:0  HMI_STATUS_ADS_A  "HMI Status word for Adsorber A" %

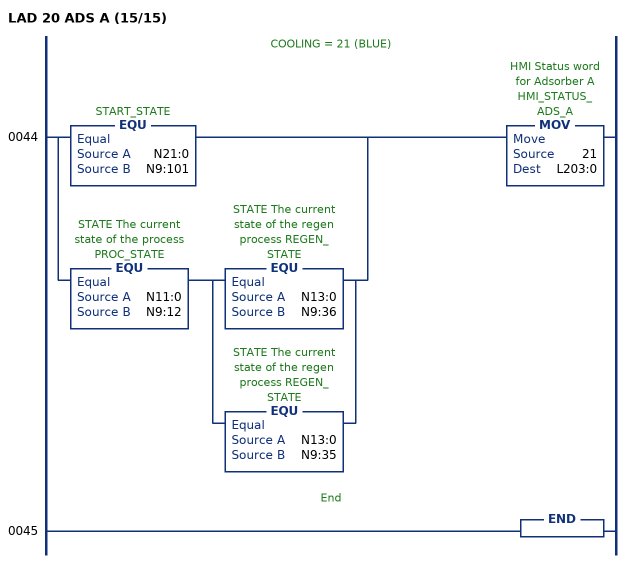
% Rung: 44 %
% COOLING = 21 (BLUE) %
SOR BST EQU N21:0 N9:101 NXB EQU N11:0 N9:12 BST EQU N13:0 N9:36 NXB EQU N13:0 N9:35 BND BND MOV 21 L203:0 EOR
%   N21:0  START_STATE %
%   N9:101  START_COOL %
%   N11:0  PROC_STATE  "STATE The current state of the process" %
%   N9:12  PROC_PFY_B_REG_A  "STATE Process Purify B" %
%   N13:0  REGEN_STATE  "STATE The current state of the regen process" %
%   N9:36  REGEN_COOL  "STATE Regen Cool" %
%   N9:35  REGEN_COOL_WALL  "STATE Regen Cool wall" %
%   L203:0  HMI_STATUS_ADS_A  "HMI Status word for Adsorber A" %
% Rung: 45 %
% End %
SOR END EOR

LADDER 21 "ADS A FLT"    % Controls the Adsorber A faults %
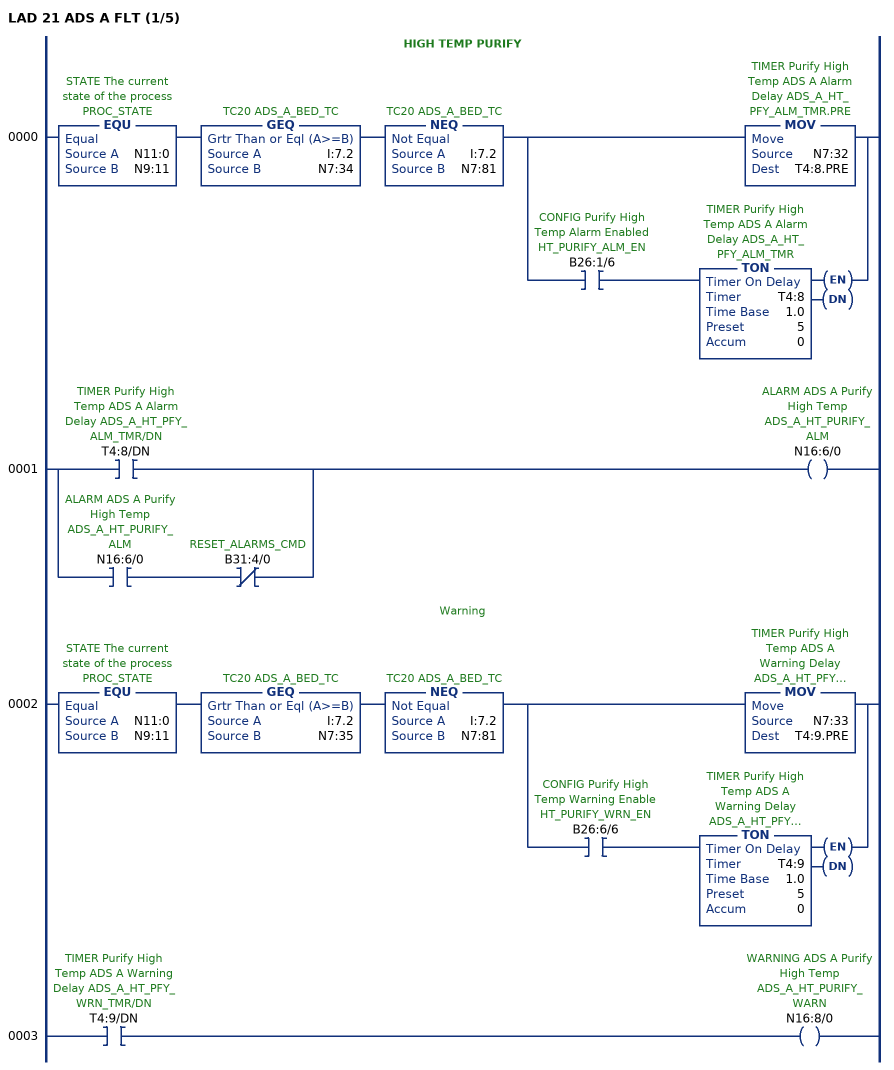
% Rung: 0 %
% TITLE: HIGH TEMP PURIFY %
SOR EQU N11:0 N9:11 GEQ I:7.2 N7:34 NEQ I:7.2 N7:81 BST MOV N7:32 T4:8.PRE NXB XIC B26:1/6 TON T4:8 1.0 5 0 BND EOR
%   N11:0  PROC_STATE  "STATE The current state of the process" %
%   N9:11  PROC_PFY_A_REG_B  "STATE Process Purify A" %
%   I:7.2  ADS_A_BED_TC  "TC20" %
%   N7:34  HT_PURIFY_ALM_SP  "CONFIG Purify High Temp Alarm Setpoint" %
%   N7:81  TC_OPEN_SP  "CONFIG The value read by an open TC input" %
%   N7:32  HT_PURIFY_ALM_DLY  "CONFIG Purify High Temp Alarm Delay" %
%   T4:8  ADS_A_HT_PFY_ALM_TMR  "TIMER Purify High Temp ADS A Alarm Delay" %
%   B26:1/6  HT_PURIFY_ALM_EN  "CONFIG Purify High Temp Alarm Enabled" %
% Rung: 1 %
SOR BST XIC T4:8/DN NXB XIC N16:6/0 XIO B31:4/0 BND OTE N16:6/0 EOR
%   T4:8  ADS_A_HT_PFY_ALM_TMR  "TIMER Purify High Temp ADS A Alarm Delay" %
%   N16:6/0  ADS_A_HT_PURIFY_ALM  "ALARM ADS A Purify High Temp" %
%   B31:4/0  RESET_ALARMS_CMD %
% Rung: 2 %
% Warning %
SOR EQU N11:0 N9:11 GEQ I:7.2 N7:35 NEQ I:7.2 N7:81 BST MOV N7:33 T4:9.PRE NXB XIC B26:6/6 TON T4:9 1.0 5 0 BND EOR
%   N11:0  PROC_STATE  "STATE The current state of the process" %
%   N9:11  PROC_PFY_A_REG_B  "STATE Process Purify A" %
%   I:7.2  ADS_A_BED_TC  "TC20" %
%   N7:35  HT_PURIFY_WRN_SP  "CONFIG Purify High Temp Warning Setpoint" %
%   N7:81  TC_OPEN_SP  "CONFIG The value read by an open TC input" %
%   N7:33  HT_PURIFY_WRN_DLY  "CONFIG Purify High Temp Warning Delay" %
%   T4:9  ADS_A_HT_PFY_WRN_TMR  "TIMER Purify High Temp ADS A Warning Delay" %
%   B26:6/6  HT_PURIFY_WRN_EN  "CONFIG Purify High Temp Warning Enable" %
% Rung: 3 %
SOR XIC T4:9/DN OTE N16:8/0 EOR
%   T4:9  ADS_A_HT_PFY_WRN_TMR  "TIMER Purify High Temp ADS A Warning Delay" %
%   N16:8/0  ADS_A_HT_PURIFY_WARN  "WARNING ADS A Purify High Temp" %

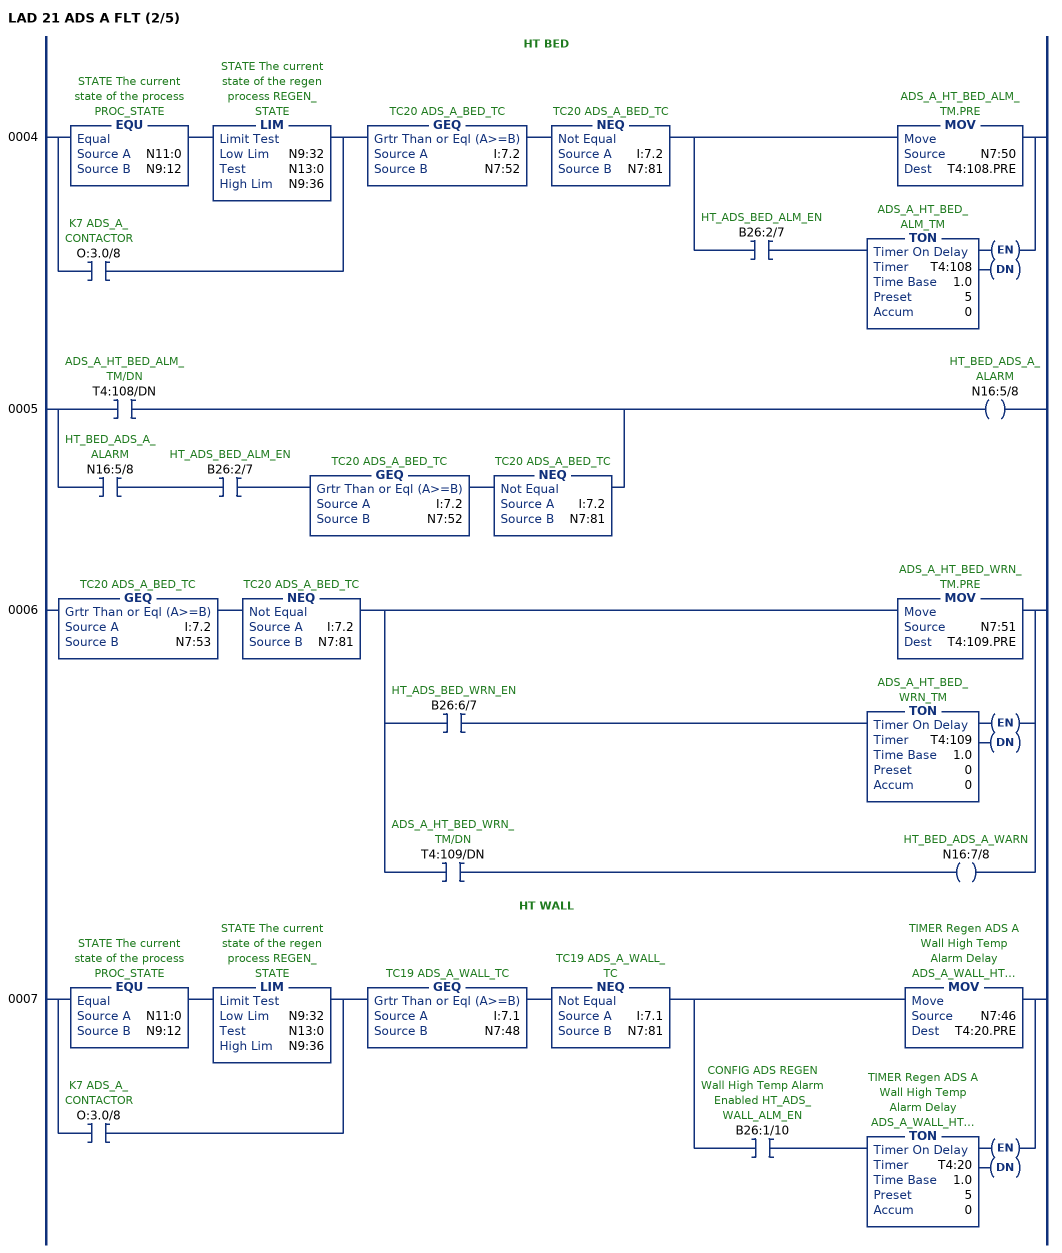
% Rung: 4 %
% TITLE: HT BED %
SOR BST EQU N11:0 N9:12 LIM N9:32 N13:0 N9:36 NXB XIC O:3.0/8 BND GEQ I:7.2 N7:52 NEQ I:7.2 N7:81 BST MOV N7:50 T4:108.PRE NXB XIC B26:2/7 TON T4:108 1.0 5 0 BND EOR
%   N11:0  PROC_STATE  "STATE The current state of the process" %
%   N9:12  PROC_PFY_B_REG_A  "STATE Process Purify B" %
%   N9:32  REGEN_VENT  "STATE Regen Vent" %
%   N13:0  REGEN_STATE  "STATE The current state of the regen process" %
%   N9:36  REGEN_COOL  "STATE Regen Cool" %
%   O:3.0/8  ADS_A_CONTACTOR  "K7" %
%   I:7.2  ADS_A_BED_TC  "TC20" %
%   N7:52  HT_ADS_BED_ALM_SP %
%   N7:81  TC_OPEN_SP  "CONFIG The value read by an open TC input" %
%   N7:50  HT_ADS_BED_ALM_DLY %
%   T4:108  ADS_A_HT_BED_ALM_TM %
%   B26:2/7  HT_ADS_BED_ALM_EN %
% Rung: 5 %
SOR BST XIC T4:108/DN NXB XIC N16:5/8 XIC B26:2/7 GEQ I:7.2 N7:52 NEQ I:7.2 N7:81 BND OTE N16:5/8 EOR
%   T4:108  ADS_A_HT_BED_ALM_TM %
%   N16:5/8  HT_BED_ADS_A_ALARM %
%   B26:2/7  HT_ADS_BED_ALM_EN %
%   I:7.2  ADS_A_BED_TC  "TC20" %
%   N7:52  HT_ADS_BED_ALM_SP %
%   N7:81  TC_OPEN_SP  "CONFIG The value read by an open TC input" %
% Rung: 6 %
SOR GEQ I:7.2 N7:53 NEQ I:7.2 N7:81 BST MOV N7:51 T4:109.PRE NXB XIC B26:6/7 TON T4:109 1.0 0 0 NXB XIC T4:109/DN OTE N16:7/8 BND EOR
%   I:7.2  ADS_A_BED_TC  "TC20" %
%   N7:53  HT_ADS_BED_WRN_SP %
%   N7:81  TC_OPEN_SP  "CONFIG The value read by an open TC input" %
%   N7:51  HT_ADS_BED_WRN_DLY %
%   T4:109  ADS_A_HT_BED_WRN_TM %
%   B26:6/7  HT_ADS_BED_WRN_EN %
%   N16:7/8  HT_BED_ADS_A_WARN %
% Rung: 7 %
% TITLE: HT WALL %
SOR BST EQU N11:0 N9:12 LIM N9:32 N13:0 N9:36 NXB XIC O:3.0/8 BND GEQ I:7.1 N7:48 NEQ I:7.1 N7:81 BST MOV N7:46 T4:20.PRE NXB XIC B26:1/10 TON T4:20 1.0 5 0 BND EOR
%   N11:0  PROC_STATE  "STATE The current state of the process" %
%   N9:12  PROC_PFY_B_REG_A  "STATE Process Purify B" %
%   N9:32  REGEN_VENT  "STATE Regen Vent" %
%   N13:0  REGEN_STATE  "STATE The current state of the regen process" %
%   N9:36  REGEN_COOL  "STATE Regen Cool" %
%   O:3.0/8  ADS_A_CONTACTOR  "K7" %
%   I:7.1  ADS_A_WALL_TC  "TC19" %
%   N7:48  HT_ADS_WALL_ALM_SP  "CONFIG ADS Wall Regen High Temp Alarm" %
%   N7:81  TC_OPEN_SP  "CONFIG The value read by an open TC input" %
%   N7:46  HT_ADS_WALL_ALM_DLY  "CONFIG ADS Wall High Temperature Alarm Delay" %
%   T4:20  ADS_A_WALL_HT_ALM_TM  "TIMER Regen ADS A Wall High Temp Alarm Delay" %
%   B26:1/10  HT_ADS_WALL_ALM_EN  "CONFIG ADS REGEN Wall High Temp Alarm Enabled" %

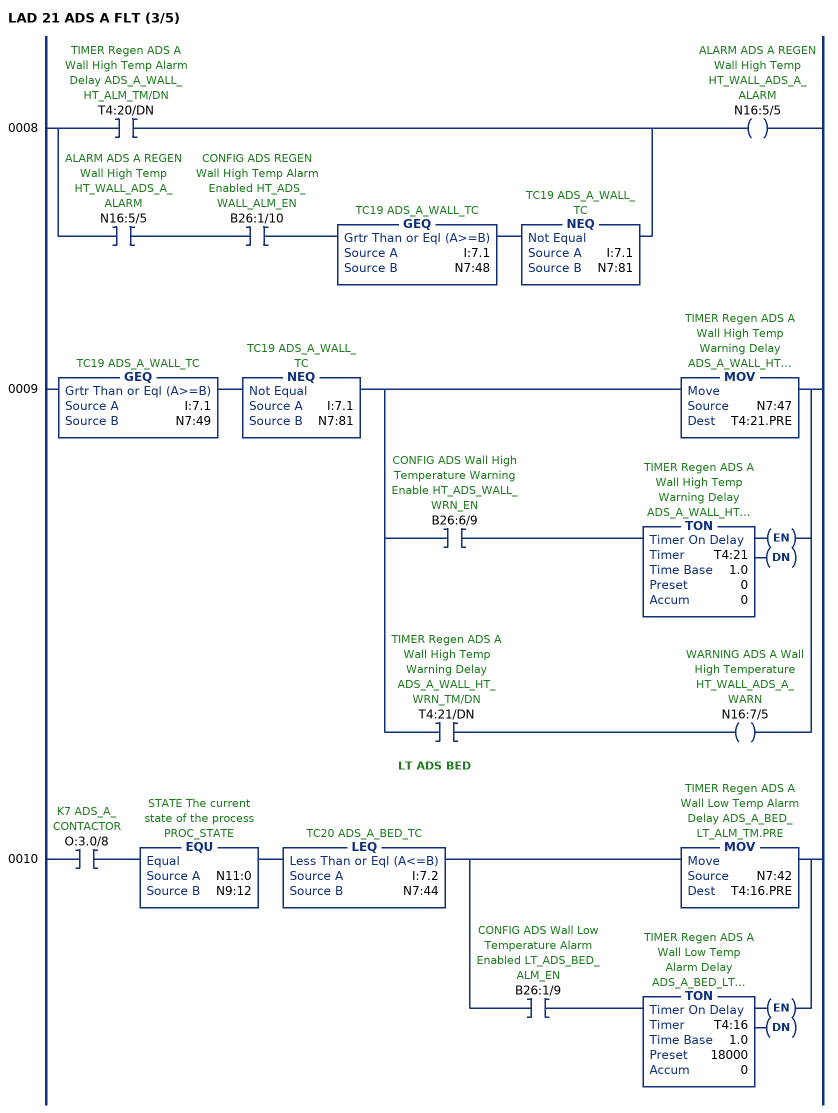
% Rung: 8 %
SOR BST XIC T4:20/DN NXB XIC N16:5/5 XIC B26:1/10 GEQ I:7.1 N7:48 NEQ I:7.1 N7:81 BND OTE N16:5/5 EOR
%   T4:20  ADS_A_WALL_HT_ALM_TM  "TIMER Regen ADS A Wall High Temp Alarm Delay" %
%   N16:5/5  HT_WALL_ADS_A_ALARM  "ALARM ADS A REGEN Wall High Temp" %
%   B26:1/10  HT_ADS_WALL_ALM_EN  "CONFIG ADS REGEN Wall High Temp Alarm Enabled" %
%   I:7.1  ADS_A_WALL_TC  "TC19" %
%   N7:48  HT_ADS_WALL_ALM_SP  "CONFIG ADS Wall Regen High Temp Alarm" %
%   N7:81  TC_OPEN_SP  "CONFIG The value read by an open TC input" %
% Rung: 9 %
SOR GEQ I:7.1 N7:49 NEQ I:7.1 N7:81 BST MOV N7:47 T4:21.PRE NXB XIC B26:6/9 TON T4:21 1.0 0 0 NXB XIC T4:21/DN OTE N16:7/5 BND EOR
%   I:7.1  ADS_A_WALL_TC  "TC19" %
%   N7:49  HT_ADS_WALL_WRN_SP  "CONFIG ADS Wall Regen High Temp Alarm" %
%   N7:81  TC_OPEN_SP  "CONFIG The value read by an open TC input" %
%   N7:47  HT_ADS_WALL_WRN_DLY  "CONFIG ADS Wall High Temperature Warning Delay" %
%   T4:21  ADS_A_WALL_HT_WRN_TM  "TIMER Regen ADS A Wall High Temp Warning Delay" %
%   B26:6/9  HT_ADS_WALL_WRN_EN  "CONFIG ADS Wall High Temperature Warning Enable" %
%   N16:7/5  HT_WALL_ADS_A_WARN  "WARNING ADS A Wall High Temperature" %
% Rung: 10 %
% TITLE: LT ADS BED %
SOR XIC O:3.0/8 EQU N11:0 N9:12 LEQ I:7.2 N7:44 BST MOV N7:42 T4:16.PRE NXB XIC B26:1/9 TON T4:16 1.0 18000 0 BND EOR
%   O:3.0/8  ADS_A_CONTACTOR  "K7" %
%   N11:0  PROC_STATE  "STATE The current state of the process" %
%   N9:12  PROC_PFY_B_REG_A  "STATE Process Purify B" %
%   I:7.2  ADS_A_BED_TC  "TC20" %
%   N7:44  LT_ADS_BED_ALM_SP  "CONFIG ADS Wall Regen Heat Low Temperature Alarm Setpoint" %
%   N7:42  LT_ADS_BED_ALM_DLY  "CONFIG ADS Wall Regen heat Low Temperature Alarm Delay" %
%   T4:16  ADS_A_BED_LT_ALM_TM  "TIMER Regen ADS A Wall Low Temp Alarm Delay" %
%   B26:1/9  LT_ADS_BED_ALM_EN  "CONFIG ADS Wall Low Temperature Alarm Enabled" %

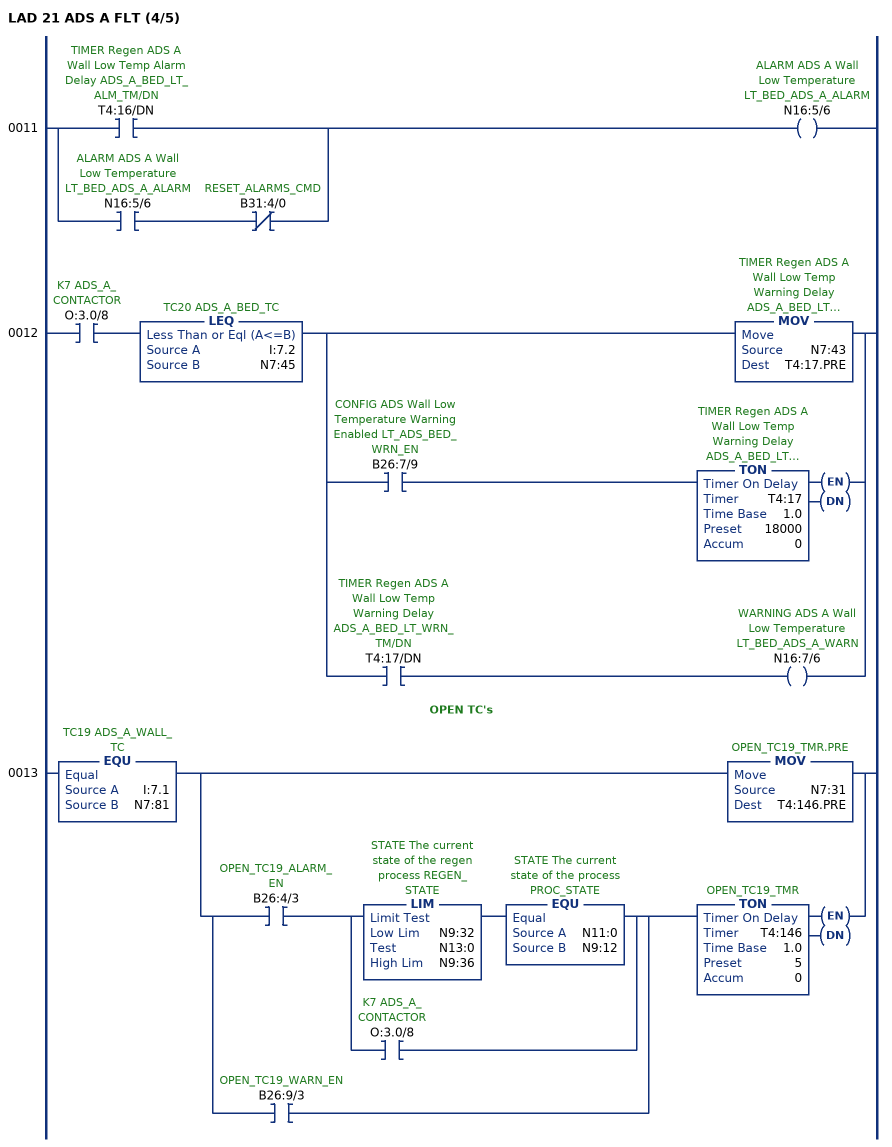
% Rung: 11 %
SOR BST XIC T4:16/DN NXB XIC N16:5/6 XIO B31:4/0 BND OTE N16:5/6 EOR
%   T4:16  ADS_A_BED_LT_ALM_TM  "TIMER Regen ADS A Wall Low Temp Alarm Delay" %
%   N16:5/6  LT_BED_ADS_A_ALARM  "ALARM ADS A Wall Low Temperature" %
%   B31:4/0  RESET_ALARMS_CMD %
% Rung: 12 %
SOR XIC O:3.0/8 LEQ I:7.2 N7:45 BST MOV N7:43 T4:17.PRE NXB XIC B26:7/9 TON T4:17 1.0 18000 0 NXB XIC T4:17/DN OTE N16:7/6 BND EOR
%   O:3.0/8  ADS_A_CONTACTOR  "K7" %
%   I:7.2  ADS_A_BED_TC  "TC20" %
%   N7:45  LT_ADS_BED_WRN_SP  "CONFIG ADS Wall Regen Heat Low Temperature Warning Setpoint" %
%   N7:43  LT_ADS_BED_WRN_DLY  "CONFIG ADS Wall Regen heat Low Temperature Warning Delay" %
%   T4:17  ADS_A_BED_LT_WRN_TM  "TIMER Regen ADS A Wall Low Temp Warning Delay" %
%   B26:7/9  LT_ADS_BED_WRN_EN  "CONFIG ADS Wall Low Temperature Warning Enabled" %
%   N16:7/6  LT_BED_ADS_A_WARN  "WARNING ADS A Wall Low Temperature" %
% Rung: 13 %
% TITLE: OPEN TC's %
SOR EQU I:7.1 N7:81 BST MOV N7:31 T4:146.PRE NXB BST XIC B26:4/3 BST LIM N9:32 N13:0 N9:36 EQU N11:0 N9:12 NXB XIC O:3.0/8 BND NXB XIC B26:9/3 BND TON T4:146 1.0 5 0 BND EOR
%   I:7.1  ADS_A_WALL_TC  "TC19" %
%   N7:81  TC_OPEN_SP  "CONFIG The value read by an open TC input" %
%   N7:31  OPEN_TC_DLY %
%   T4:146  OPEN_TC19_TMR %
%   B26:4/3  OPEN_TC19_ALARM_EN %
%   N9:32  REGEN_VENT  "STATE Regen Vent" %
%   N13:0  REGEN_STATE  "STATE The current state of the regen process" %
%   N9:36  REGEN_COOL  "STATE Regen Cool" %
%   N11:0  PROC_STATE  "STATE The current state of the process" %
%   N9:12  PROC_PFY_B_REG_A  "STATE Process Purify B" %
%   O:3.0/8  ADS_A_CONTACTOR  "K7" %
%   B26:9/3  OPEN_TC19_WARN_EN %

